LIN {X 0,Y 239.428,Z 683.696,A -85,B 0,C 180,E1 8082.611,E2 8082.611} C_VEL
LIN {X 0,Y 240.054,Z 699.149,A -85,B 0,C 180,E1 8081.155,E2 8081.155} C_VEL
LIN {X 0,Y 233.053,Z 774.476,A -85,B 0,C 180,E1 8079.078,E2 8079.078} C_VEL
LIN {X 0,Y 230.461,Z 791.009,A -85,B 0,C 180,E1 8078.257,E2 8078.257} C_VEL
LIN {X 0,Y 226.592,Z 807.31,A -85,B 0,C 180,E1 8077.072,E2 8077.072} C_VEL
LIN {X 0,Y 221.78,Z 822.279,A -85,B 0,C 180,E1 8075.581,E2 8075.581} C_VEL
LIN {X 0,Y 215.863,Z 836.74,A -85,B 0,C 180,E1 8073.655,E2 8073.655} C_VEL
LIN {X 0,Y 209.493,Z 849.592,A -85,B 0,C 180,E1 8071.408,E2 8071.408} C_VEL
LIN {X 0,Y 202.485,Z 861.469,A -85,B 0,C 180,E1 8068.664,E2 8068.664} C_VEL
LIN {X 0,Y 195.095,Z 872.265,A -85,B 0,C 180,E1 8065.327,E2 8065.327} C_VEL
LIN {X 0,Y 188.35,Z 880.818,A -85,B 0,C 180,E1 8061.77,E2 8061.77} C_VEL
LIN {X 0,Y 181.644,Z 888.195,A -85,B 0,C 180,E1 8057.516,E2 8057.516} C_VEL
LIN {X 0,Y 175.57,Z 894.029,A -85,B 0,C 180,E1 8052.654,E2 8052.654} C_VEL
LIN {X 0,Y 170.723,Z 897.867,A -85,B 0,C 180,E1 8047.515,E2 8047.515} C_VEL
LIN {X 0,Y 166.949,Z 900.056,A -85,B 0,C 180,E1 8041.739,E2 8041.739} C_VEL
LIN {X 0,Y 164.662,Z 900.334,A -85,B 0,C 180,E1 8035.918,E2 8035.918} C_VEL
LIN {X 0,Y 163.665,Z 898.731,A -85,B 0,C 180,E1 8029.809,E2 8029.809} C_VEL
LIN {X 0,Y 163.914,Z 895.477,A -85,B 0,C 180,E1 8024.093,E2 8024.093} C_VEL
LIN {X 0,Y 165.328,Z 890.237,A -85,B 0,C 180,E1 8018.341,E2 8018.341} C_VEL
LIN {X 0,Y 167.764,Z 883.453,A -85,B 0,C 180,E1 8013.07,E2 8013.07} C_VEL
LIN {X 0,Y 171.056,Z 875.039,A -85,B 0,C 180,E1 8008.273,E2 8008.273} C_VEL
LIN {X 0,Y 174.923,Z 865.341,A -85,B 0,C 180,E1 8004.041,E2 8004.041} C_VEL
LIN {X 0,Y 179.081,Z 854.36,A -85,B 0,C 180,E1 8000.354,E2 8000.354} C_VEL
LIN {X 0,Y 183.652,Z 841.158,A -85,B 0,C 180,E1 7996.939,E2 7996.939} C_VEL
LIN {X 0,Y 187.804,Z 827.496,A -85,B 0,C 180,E1 7994.243,E2 7994.243} C_VEL
LIN {X 0,Y 191.755,Z 811.933,A -85,B 0,C 180,E1 7991.924,E2 7991.924} C_VEL
LIN {X 0,Y 194.868,Z 796.193,A -85,B 0,C 180,E1 7990.204,E2 7990.204} C_VEL
LIN {X 0,Y 197.282,Z 778.863,A -85,B 0,C 180,E1 7988.888,E2 7988.888} C_VEL
LIN {X 0,Y 198.697,Z 760.857,A -85,B 0,C 180,E1 7988.063,E2 7988.063} C_VEL
LIN {X 0,Y 203.572,Z 686.601,A -85,B 0,C 180,E1 7985.632,E2 7985.632} C_VEL
LIN {X 0,Y 199.817,Z 646.699,A -85,B 0,C 180,E1 7982.617,E2 7982.617} C_VEL
LIN {X 0,Y 192.297,Z 631.171,A -85,B 0,C 180,E1 7979.45,E2 7979.45} C_VEL
LIN {X 0,Y 189.561,Z 625.909,A -85,B 0,C 180,E1 7978.127,E2 7978.127} C_VEL
LIN {X 0,Y 187.323,Z 616.123,A -85,B 0,C 180,E1 7973.193,E2 7973.193} C_VEL
LIN {X 0,Y 184.89,Z 607.378,A -85,B 0,C 180,E1 7967.888,E2 7967.888} C_VEL
LIN {X 0,Y 182.856,Z 600.739,A -85,B 0,C 180,E1 7963.119,E2 7963.119} C_VEL
LIN {X 0,Y 180.838,Z 594.707,A -85,B 0,C 180,E1 7957.86,E2 7957.86} C_VEL
LIN {X 0,Y 179.177,Z 590.553,A -85,B 0,C 180,E1 7953.153,E2 7953.153} C_VEL
LIN {X 0,Y 177.959,Z 587.255,A -85,B 0,C 180,E1 7948.528,E2 7948.528} C_VEL
LIN {X 0,Y 176.637,Z 583.641,A -85,B 0,C 180,E1 7940.546,E2 7940.546} C_VEL
LIN {X 0,Y 176.092,Z 582.922,A -85,B 0,C 180,E1 7934.133,E2 7934.133} C_VEL
LIN {X 0,Y 176.584,Z 583.469,A -85,B 0,C 180,E1 7927.484,E2 7927.484} C_VEL
LIN {X 0,Y 177.159,Z 584.592,A -85,B 0,C 180,E1 7923.884,E2 7923.884} C_VEL
LIN {X 0,Y 179.034,Z 588.581,A -85,B 0,C 180,E1 7916.479,E2 7916.479} C_VEL
LIN {X 0,Y 180.799,Z 592.823,A -85,B 0,C 180,E1 7911.413,E2 7911.413} C_VEL
LIN {X 0,Y 182.534,Z 597.114,A -85,B 0,C 180,E1 7907.344,E2 7907.344} C_VEL
LIN {X 0,Y 185.067,Z 603.482,A -85,B 0,C 180,E1 7902.39,E2 7902.39} C_VEL
LIN {X 0,Y 188.02,Z 611.83,A -85,B 0,C 180,E1 7897.158,E2 7897.158} C_VEL
LIN {X 0,Y 191.069,Z 621.45,A -85,B 0,C 180,E1 7892.243,E2 7892.243} C_VEL
LIN {X 0,Y 198.28,Z 634.127,A -85,B 0,C 180,E1 7889.131,E2 7889.131} C_VEL
LIN {X 0,Y 205.837,Z 648.788,A -85,B 0,C 180,E1 7886.25,E2 7886.25} C_VEL
LIN {X 0,Y 208.597,Z 655.147,A -85,B 0,C 180,E1 7885.223,E2 7885.223} C_VEL
LIN {X 0,Y 208.82,Z 667.164,A -85,B 0,C 180,E1 7884.604,E2 7884.604} C_VEL
LIN {X 0,Y 203.561,Z 748.117,A -85,B 0,C 180,E1 7882.187,E2 7882.187} C_VEL
LIN {X 0,Y 202.351,Z 755.783,A -85,B 0,C 180,E1 7882.134,E2 7882.134} C_VEL
LIN {X 0,Y 196.3,Z 776.069,A -85,B 0,C 180,E1 7882.677,E2 7882.677} C_VEL
LIN {X 0,Y 195.302,Z 782.654,A -85,B 0,C 180,E1 7882.62,E2 7882.62} C_VEL
LIN {X 0,Y 193.611,Z 802.35,A -85,B 0,C 180,E1 7881.852,E2 7881.852} C_VEL
LIN {X 0,Y 190.848,Z 819.979,A -85,B 0,C 180,E1 7880.72,E2 7880.72} C_VEL
LIN {X 0,Y 186.92,Z 837.364,A -85,B 0,C 180,E1 7879.124,E2 7879.124} C_VEL
LIN {X 0,Y 182.366,Z 853.624,A -85,B 0,C 180,E1 7877.058,E2 7877.058} C_VEL
LIN {X 0,Y 177.233,Z 869.3,A -85,B 0,C 180,E1 7874.391,E2 7874.391} C_VEL
LIN {X 0,Y 171.883,Z 883.863,A -85,B 0,C 180,E1 7871.098,E2 7871.098} C_VEL
LIN {X 0,Y 166.529,Z 897.391,A -85,B 0,C 180,E1 7867.116,E2 7867.116} C_VEL
LIN {X 0,Y 161.793,Z 909.403,A -85,B 0,C 180,E1 7862.526,E2 7862.526} C_VEL
LIN {X 0,Y 158.011,Z 919.598,A -85,B 0,C 180,E1 7857.514,E2 7857.514} C_VEL
LIN {X 0,Y 155.289,Z 928.39,A -85,B 0,C 180,E1 7851.931,E2 7851.931} C_VEL
LIN {X 0,Y 153.926,Z 935.715,A -85,B 0,C 180,E1 7845.835,E2 7845.835} C_VEL
LIN {X 0,Y 154.037,Z 941.459,A -85,B 0,C 180,E1 7839.343,E2 7839.343} C_VEL
LIN {X 0,Y 155.114,Z 944.871,A -85,B 0,C 180,E1 7833.7,E2 7833.7} C_VEL
LIN {X 0,Y 155.742,Z 946.247,A -85,B 0,C 180,E1 7830.004,E2 7830.004} C_VEL
LIN {X 0,Y 154.8,Z 946.748,A -85,B 0,C 180,E1 7825.931,E2 7825.931} C_VEL
LIN {X 0,Y 153.503,Z 945.982,A -85,B 0,C 180,E1 7819.497,E2 7819.497} C_VEL
LIN {X 0,Y 153.729,Z 943.404,A -85,B 0,C 180,E1 7812.598,E2 7812.598} C_VEL
LIN {X 0,Y 155.999,Z 939.047,A -85,B 0,C 180,E1 7805.79,E2 7805.79} C_VEL
LIN {X 0,Y 160.423,Z 932.831,A -85,B 0,C 180,E1 7799.272,E2 7799.272} C_VEL
LIN {X 0,Y 166.479,Z 925.115,A -85,B 0,C 180,E1 7793.526,E2 7793.526} C_VEL
LIN {X 0,Y 173.691,Z 915.929,A -85,B 0,C 180,E1 7788.557,E2 7788.557} C_VEL
LIN {X 0,Y 181.69,Z 905.294,A -85,B 0,C 180,E1 7784.334,E2 7784.334} C_VEL
LIN {X 0,Y 190.524,Z 892.551,A -85,B 0,C 180,E1 7780.597,E2 7780.597} C_VEL
LIN {X 0,Y 198.904,Z 879.059,A -85,B 0,C 180,E1 7777.665,E2 7777.665} C_VEL
LIN {X 0,Y 206.592,Z 864.904,A -85,B 0,C 180,E1 7775.376,E2 7775.376} C_VEL
LIN {X 0,Y 213.561,Z 849.877,A -85,B 0,C 180,E1 7773.567,E2 7773.567} C_VEL
LIN {X 0,Y 219.656,Z 834.019,A -85,B 0,C 180,E1 7772.164,E2 7772.164} C_VEL
LIN {X 0,Y 224.755,Z 817.067,A -85,B 0,C 180,E1 7771.078,E2 7771.078} C_VEL
LIN {X 0,Y 228.519,Z 799.346,A -85,B 0,C 180,E1 7770.277,E2 7770.277} C_VEL
LIN {X 0,Y 230.844,Z 779.683,A -85,B 0,C 180,E1 7769.691,E2 7769.691} C_VEL
LIN {X 0,Y 239.232,Z 685.969,A -85,B 0,C 180,E1 7767.302,E2 7767.302} C_VEL
LIN {X 0,Y 234.919,Z 677.468,A -85,B 0,C 180,E1 7764.116,E2 7764.116} C_VEL
LIN {X 0,Y 231.392,Z 671.367,A -85,B 0,C 180,E1 7761.017,E2 7761.017} C_VEL
LIN {X 0,Y 228.729,Z 667.122,A -85,B 0,C 180,E1 7758.213,E2 7758.213} C_VEL
LIN {X 0,Y 226.198,Z 663.254,A -85,B 0,C 180,E1 7754.724,E2 7754.724} C_VEL
LIN {X 0,Y 224.164,Z 660.314,A -85,B 0,C 180,E1 7750.537,E2 7750.537} C_VEL
LIN {X 0,Y 223.09,Z 659.552,A -85,B 0,C 180,E1 7744.884,E2 7744.884} C_VEL
LIN {X 0,Y 223.271,Z 660.346,A -85,B 0,C 180,E1 7742.309,E2 7742.309} C_VEL
LIN {X 0,Y 224.694,Z 663.258,A -85,B 0,C 180,E1 7737.449,E2 7737.449} C_VEL
LIN {X 0,Y 227.153,Z 668.305,A -85,B 0,C 180,E1 7733.174,E2 7733.174} C_VEL
LIN {X 0,Y 229.056,Z 672.328,A -85,B 0,C 180,E1 7730.705,E2 7730.705} C_VEL
LIN {X 0,Y 231.536,Z 677.558,A -85,B 0,C 180,E1 7728.1,E2 7728.1} C_VEL
LIN {X 0,Y 234.13,Z 683.469,A -85,B 0,C 180,E1 7725.722,E2 7725.722} C_VEL
LIN {X 0,Y 236.21,Z 688.871,A -85,B 0,C 180,E1 7723.982,E2 7723.982} C_VEL
LIN {X 0,Y 236.518,Z 700.902,A -85,B 0,C 180,E1 7722.858,E2 7722.858} C_VEL
LIN {X 0,Y 229.387,Z 775.054,A -85,B 0,C 180,E1 7720.834,E2 7720.834} C_VEL
LIN {X 0,Y 226.705,Z 791.601,A -85,B 0,C 180,E1 7720.023,E2 7720.023} C_VEL
LIN {X 0,Y 222.69,Z 807.951,A -85,B 0,C 180,E1 7718.85,E2 7718.85} C_VEL
LIN {X 0,Y 217.695,Z 822.98,A -85,B 0,C 180,E1 7717.375,E2 7717.375} C_VEL
LIN {X 0,Y 211.543,Z 837.477,A -85,B 0,C 180,E1 7715.465,E2 7715.465} C_VEL
LIN {X 0,Y 204.564,Z 850.981,A -85,B 0,C 180,E1 7713.11,E2 7713.11} C_VEL
LIN {X 0,Y 197.162,Z 862.876,A -85,B 0,C 180,E1 7710.331,E2 7710.331} C_VEL
LIN {X 0,Y 189.505,Z 873.477,A -85,B 0,C 180,E1 7707.011,E2 7707.011} C_VEL
LIN {X 0,Y 182.068,Z 882.342,A -85,B 0,C 180,E1 7703.23,E2 7703.23} C_VEL
LIN {X 0,Y 175.061,Z 889.586,A -85,B 0,C 180,E1 7698.919,E2 7698.919} C_VEL
LIN {X 0,Y 168.617,Z 895.358,A -85,B 0,C 180,E1 7693.92,E2 7693.92} C_VEL
LIN {X 0,Y 163.251,Z 899.255,A -85,B 0,C 180,E1 7688.374,E2 7688.374} C_VEL
LIN {X 0,Y 159.396,Z 901.278,A -85,B 0,C 180,E1 7682.639,E2 7682.639} C_VEL
LIN {X 0,Y 156.986,Z 901.582,A -85,B 0,C 180,E1 7676.878,E2 7676.878} C_VEL
LIN {X 0,Y 155.776,Z 900.032,A -85,B 0,C 180,E1 7670.425,E2 7670.425} C_VEL
LIN {X 0,Y 155.924,Z 896.909,A -85,B 0,C 180,E1 7664.465,E2 7664.465} C_VEL
LIN {X 0,Y 157.191,Z 892.148,A -85,B 0,C 180,E1 7658.776,E2 7658.776} C_VEL
LIN {X 0,Y 159.593,Z 885.6,A -85,B 0,C 180,E1 7653.228,E2 7653.228} C_VEL
LIN {X 0,Y 162.875,Z 877.634,A -85,B 0,C 180,E1 7648.237,E2 7648.237} C_VEL
LIN {X 0,Y 167.129,Z 867.453,A -85,B 0,C 180,E1 7643.47,E2 7643.47} C_VEL
LIN {X 0,Y 171.691,Z 856.124,A -85,B 0,C 180,E1 7639.426,E2 7639.426} C_VEL
LIN {X 0,Y 176.451,Z 843.081,A -85,B 0,C 180,E1 7635.895,E2 7635.895} C_VEL
LIN {X 0,Y 180.761,Z 829.784,A -85,B 0,C 180,E1 7633.126,E2 7633.126} C_VEL
LIN {X 0,Y 184.887,Z 814.509,A -85,B 0,C 180,E1 7630.736,E2 7630.736} C_VEL
LIN {X 0,Y 188.268,Z 798.796,A -85,B 0,C 180,E1 7628.91,E2 7628.91} C_VEL
LIN {X 0,Y 190.822,Z 781.973,A -85,B 0,C 180,E1 7627.55,E2 7627.55} C_VEL
LIN {X 0,Y 192.42,Z 764.7,A -85,B 0,C 180,E1 7626.667,E2 7626.667} C_VEL
LIN {X 0,Y 197.669,Z 687.648,A -85,B 0,C 180,E1 7624.1,E2 7624.1} C_VEL
LIN {X 0,Y 194.418,Z 650.352,A -85,B 0,C 180,E1 7621.19,E2 7621.19} C_VEL
LIN {X 0,Y 187.727,Z 636.24,A -85,B 0,C 180,E1 7618.161,E2 7618.161} C_VEL
LIN {X 0,Y 182.096,Z 625.601,A -85,B 0,C 180,E1 7615.284,E2 7615.284} C_VEL
LIN {X 0,Y 180.173,Z 617.536,A -85,B 0,C 180,E1 7610.754,E2 7610.754} C_VEL
LIN {X 0,Y 178.21,Z 610.241,A -85,B 0,C 180,E1 7605.903,E2 7605.903} C_VEL
LIN {X 0,Y 176.352,Z 604.108,A -85,B 0,C 180,E1 7601.056,E2 7601.056} C_VEL
LIN {X 0,Y 174.761,Z 599.428,A -85,B 0,C 180,E1 7596.514,E2 7596.514} C_VEL
LIN {X 0,Y 173.64,Z 596.234,A -85,B 0,C 180,E1 7592.771,E2 7592.771} C_VEL
LIN {X 0,Y 172.573,Z 593.132,A -85,B 0,C 180,E1 7588.278,E2 7588.278} C_VEL
LIN {X 0,Y 171.434,Z 589.715,A -85,B 0,C 180,E1 7580.484,E2 7580.484} C_VEL
LIN {X 0,Y 170.944,Z 589.036,A -85,B 0,C 180,E1 7573.85,E2 7573.85} C_VEL
LIN {X 0,Y 171.464,Z 589.628,A -85,B 0,C 180,E1 7567.371,E2 7567.371} C_VEL
LIN {X 0,Y 171.97,Z 590.687,A -85,B 0,C 180,E1 7564.001,E2 7564.001} C_VEL
LIN {X 0,Y 173.71,Z 594.549,A -85,B 0,C 180,E1 7556.701,E2 7556.701} C_VEL
LIN {X 0,Y 175.407,Z 598.878,A -85,B 0,C 180,E1 7551.478,E2 7551.478} C_VEL
LIN {X 0,Y 176.998,Z 602.87,A -85,B 0,C 180,E1 7547.605,E2 7547.605} C_VEL
LIN {X 0,Y 179.299,Z 608.874,A -85,B 0,C 180,E1 7542.81,E2 7542.81} C_VEL
LIN {X 0,Y 182.117,Z 617.308,A -85,B 0,C 180,E1 7537.399,E2 7537.399} C_VEL
LIN {X 0,Y 183.778,Z 622.203,A -85,B 0,C 180,E1 7534.847,E2 7534.847} C_VEL
LIN {X 0,Y 190.897,Z 634.308,A -85,B 0,C 180,E1 7531.492,E2 7531.492} C_VEL
LIN {X 0,Y 198.02,Z 647.764,A -85,B 0,C 180,E1 7528.494,E2 7528.494} C_VEL
LIN {X 0,Y 202.815,Z 658.233,A -85,B 0,C 180,E1 7526.602,E2 7526.602} C_VEL
LIN {X 0,Y 202.909,Z 668.079,A -85,B 0,C 180,E1 7526.097,E2 7526.097} C_VEL
LIN {X 0,Y 195.302,Z 782.654,A -85,B 0,C 180,E1 7522.62,E2 7522.62} C_VEL
LIN {X 0,Y 193.966,Z 790.299,A -85,B 0,C 180,E1 7522.569,E2 7522.569} C_VEL
LIN {X 0,Y 187.888,Z 807.129,A -85,B 0,C 180,E1 7522.822,E2 7522.822} C_VEL
LIN {X 0,Y 185.613,Z 814.554,A -85,B 0,C 180,E1 7522.604,E2 7522.604} C_VEL
LIN {X 0,Y 185.173,Z 816.696,A -85,B 0,C 180,E1 7522.471,E2 7522.471} C_VEL
LIN {X 0,Y 181.426,Z 833.575,A -85,B 0,C 180,E1 7520.993,E2 7520.993} C_VEL
LIN {X 0,Y 176.881,Z 849.68,A -85,B 0,C 180,E1 7519.027,E2 7519.027} C_VEL
LIN {X 0,Y 171.432,Z 866.024,A -85,B 0,C 180,E1 7516.321,E2 7516.321} C_VEL
LIN {X 0,Y 165.984,Z 880.498,A -85,B 0,C 180,E1 7513.135,E2 7513.135} C_VEL
LIN {X 0,Y 160.473,Z 893.91,A -85,B 0,C 180,E1 7509.263,E2 7509.263} C_VEL
LIN {X 0,Y 155.217,Z 906.376,A -85,B 0,C 180,E1 7504.534,E2 7504.534} C_VEL
LIN {X 0,Y 150.738,Z 917.592,A -85,B 0,C 180,E1 7498.964,E2 7498.964} C_VEL
LIN {X 0,Y 147.585,Z 926.935,A -85,B 0,C 180,E1 7492.874,E2 7492.874} C_VEL
LIN {X 0,Y 146.01,Z 934.479,A -85,B 0,C 180,E1 7486.309,E2 7486.309} C_VEL
LIN {X 0,Y 146.075,Z 940.247,A -85,B 0,C 180,E1 7479.459,E2 7479.459} C_VEL
LIN {X 0,Y 147.236,Z 943.726,A -85,B 0,C 180,E1 7473.396,E2 7473.396} C_VEL
LIN {X 0,Y 147.844,Z 944.945,A -85,B 0,C 180,E1 7470.005,E2 7470.005} C_VEL
LIN {X 0,Y 146.798,Z 945.483,A -85,B 0,C 180,E1 7465.708,E2 7465.708} C_VEL
LIN {X 0,Y 145.507,Z 944.797,A -85,B 0,C 180,E1 7458.913,E2 7458.913} C_VEL
LIN {X 0,Y 145.924,Z 942.317,A -85,B 0,C 180,E1 7451.635,E2 7451.635} C_VEL
LIN {X 0,Y 148.597,Z 937.956,A -85,B 0,C 180,E1 7444.373,E2 7444.373} C_VEL
LIN {X 0,Y 153.745,Z 931.538,A -85,B 0,C 180,E1 7437.34,E2 7437.34} C_VEL
LIN {X 0,Y 160.388,Z 923.803,A -85,B 0,C 180,E1 7431.445,E2 7431.445} C_VEL
LIN {X 0,Y 168.168,Z 914.58,A -85,B 0,C 180,E1 7426.405,E2 7426.405} C_VEL
LIN {X 0,Y 176.691,Z 903.905,A -85,B 0,C 180,E1 7422.169,E2 7422.169} C_VEL
LIN {X 0,Y 185.532,Z 891.794,A -85,B 0,C 180,E1 7418.621,E2 7418.621} C_VEL
LIN {X 0,Y 194.07,Z 878.728,A -85,B 0,C 180,E1 7415.775,E2 7415.775} C_VEL
LIN {X 0,Y 202.41,Z 864.08,A -85,B 0,C 180,E1 7413.417,E2 7413.417} C_VEL
LIN {X 0,Y 209.646,Z 849.014,A -85,B 0,C 180,E1 7411.642,E2 7411.642} C_VEL
LIN {X 0,Y 216.304,Z 832.104,A -85,B 0,C 180,E1 7410.2,E2 7410.2} C_VEL
LIN {X 0,Y 221.507,Z 814.966,A -85,B 0,C 180,E1 7409.155,E2 7409.155} C_VEL
LIN {X 0,Y 225.181,Z 797.447,A -85,B 0,C 180,E1 7408.407,E2 7408.407} C_VEL
LIN {X 0,Y 227.613,Z 776.617,A -85,B 0,C 180,E1 7407.814,E2 7407.814} C_VEL
LIN {X 0,Y 235.634,Z 690.369,A -85,B 0,C 180,E1 7405.646,E2 7405.646} C_VEL
LIN {X 0,Y 232.101,Z 683.326,A -85,B 0,C 180,E1 7402.745,E2 7402.745} C_VEL
LIN {X 0,Y 229.499,Z 678.565,A -85,B 0,C 180,E1 7400.264,E2 7400.264} C_VEL
LIN {X 0,Y 227.206,Z 674.687,A -85,B 0,C 180,E1 7397.676,E2 7397.676} C_VEL
LIN {X 0,Y 224.807,Z 670.838,A -85,B 0,C 180,E1 7394.159,E2 7394.159} C_VEL
LIN {X 0,Y 223.066,Z 668.204,A -85,B 0,C 180,E1 7390.328,E2 7390.328} C_VEL
LIN {X 0,Y 222.072,Z 667.487,A -85,B 0,C 180,E1 7384.907,E2 7384.907} C_VEL
LIN {X 0,Y 222.245,Z 668.339,A -85,B 0,C 180,E1 7382.32,E2 7382.32} C_VEL
LIN {X 0,Y 223.477,Z 671.041,A -85,B 0,C 180,E1 7377.82,E2 7377.82} C_VEL
LIN {X 0,Y 225.984,Z 676.519,A -85,B 0,C 180,E1 7373.266,E2 7373.266} C_VEL
LIN {X 0,Y 229.211,Z 683.798,A -85,B 0,C 180,E1 7369.252,E2 7369.252} C_VEL
LIN {X 0,Y 231.879,Z 690.276,A -85,B 0,C 180,E1 7366.598,E2 7366.598} C_VEL
LIN {X 0,Y 233.168,Z 694.083,A -85,B 0,C 180,E1 7365.392,E2 7365.392} C_VEL
LIN {X 0,Y 233.222,Z 702.547,A -85,B 0,C 180,E1 7364.616,E2 7364.616} C_VEL
LIN {X 0,Y 225.919,Z 775.846,A -85,B 0,C 180,E1 7362.638,E2 7362.638} C_VEL
LIN {X 0,Y 223.123,Z 792.417,A -85,B 0,C 180,E1 7361.834,E2 7361.834} C_VEL
LIN {X 0,Y 219.01,Z 808.593,A -85,B 0,C 180,E1 7360.691,E2 7360.691} C_VEL
LIN {X 0,Y 213.833,Z 823.681,A -85,B 0,C 180,E1 7359.235,E2 7359.235} C_VEL
LIN {X 0,Y 207.815,Z 837.452,A -85,B 0,C 180,E1 7357.462,E2 7357.462} C_VEL
LIN {X 0,Y 200.533,Z 851.132,A -85,B 0,C 180,E1 7355.136,E2 7355.136} C_VEL
LIN {X 0,Y 192.876,Z 863.101,A -85,B 0,C 180,E1 7352.414,E2 7352.414} C_VEL
LIN {X 0,Y 184.641,Z 874.043,A -85,B 0,C 180,E1 7349.039,E2 7349.039} C_VEL
LIN {X 0,Y 176.614,Z 883.204,A -85,B 0,C 180,E1 7345.159,E2 7345.159} C_VEL
LIN {X 0,Y 169.074,Z 890.559,A -85,B 0,C 180,E1 7340.744,E2 7340.744} C_VEL
LIN {X 0,Y 162.169,Z 896.359,A -85,B 0,C 180,E1 7335.648,E2 7335.648} C_VEL
LIN {X 0,Y 156.541,Z 900.223,A -85,B 0,C 180,E1 7330.163,E2 7330.163} C_VEL
LIN {X 0,Y 152.077,Z 902.425,A -85,B 0,C 180,E1 7323.967,E2 7323.967} C_VEL
LIN {X 0,Y 149.222,Z 902.777,A -85,B 0,C 180,E1 7317.53,E2 7317.53} C_VEL
LIN {X 0,Y 147.892,Z 901.292,A -85,B 0,C 180,E1 7310.99,E2 7310.99} C_VEL
LIN {X 0,Y 147.981,Z 898.065,A -85,B 0,C 180,E1 7304.471,E2 7304.471} C_VEL
LIN {X 0,Y 149.299,Z 893.282,A -85,B 0,C 180,E1 7298.467,E2 7298.467} C_VEL
LIN {X 0,Y 151.823,Z 886.728,A -85,B 0,C 180,E1 7292.637,E2 7292.637} C_VEL
LIN {X 0,Y 155.28,Z 878.768,A -85,B 0,C 180,E1 7287.412,E2 7287.412} C_VEL
LIN {X 0,Y 159.755,Z 868.601,A -85,B 0,C 180,E1 7282.444,E2 7282.444} C_VEL
LIN {X 0,Y 164.546,Z 857.31,A -85,B 0,C 180,E1 7278.251,E2 7278.251} C_VEL
LIN {X 0,Y 169.536,Z 844.313,A -85,B 0,C 180,E1 7274.607,E2 7274.607} C_VEL
LIN {X 0,Y 174.306,Z 830.259,A -85,B 0,C 180,E1 7271.607,E2 7271.607} C_VEL
LIN {X 0,Y 178.532,Z 815.274,A -85,B 0,C 180,E1 7269.221,E2 7269.221} C_VEL
LIN {X 0,Y 182.019,Z 799.792,A -85,B 0,C 180,E1 7267.384,E2 7267.384} C_VEL
LIN {X 0,Y 184.711,Z 783,A -85,B 0,C 180,E1 7265.992,E2 7265.992} C_VEL
LIN {X 0,Y 186.42,Z 765.577,A -85,B 0,C 180,E1 7265.077,E2 7265.077} C_VEL
LIN {X 0,Y 191.894,Z 688.725,A -85,B 0,C 180,E1 7262.487,E2 7262.487} C_VEL
LIN {X 0,Y 189.113,Z 653.977,A -85,B 0,C 180,E1 7259.67,E2 7259.67} C_VEL
LIN {X 0,Y 183.183,Z 641.172,A -85,B 0,C 180,E1 7256.772,E2 7256.772} C_VEL
LIN {X 0,Y 177.12,Z 629.878,A -85,B 0,C 180,E1 7253.556,E2 7253.556} C_VEL
LIN {X 0,Y 174.72,Z 625.277,A -85,B 0,C 180,E1 7252.014,E2 7252.014} C_VEL
LIN {X 0,Y 172.617,Z 616.63,A -85,B 0,C 180,E1 7246.39,E2 7246.39} C_VEL
LIN {X 0,Y 170.67,Z 609.919,A -85,B 0,C 180,E1 7241.008,E2 7241.008} C_VEL
LIN {X 0,Y 169.18,Z 605.096,A -85,B 0,C 180,E1 7236.229,E2 7236.229} C_VEL
LIN {X 0,Y 168.116,Z 601.918,A -85,B 0,C 180,E1 7232.363,E2 7232.363} C_VEL
LIN {X 0,Y 167.151,Z 598.936,A -85,B 0,C 180,E1 7227.813,E2 7227.813} C_VEL
LIN {X 0,Y 166.189,Z 595.721,A -85,B 0,C 180,E1 7220.057,E2 7220.057} C_VEL
LIN {X 0,Y 165.791,Z 595.169,A -85,B 0,C 180,E1 7213.249,E2 7213.249} C_VEL
LIN {X 0,Y 166.394,Z 595.862,A -85,B 0,C 180,E1 7206.903,E2 7206.903} C_VEL
LIN {X 0,Y 166.809,Z 596.944,A -85,B 0,C 180,E1 7203.781,E2 7203.781} C_VEL
LIN {X 0,Y 168.383,Z 600.51,A -85,B 0,C 180,E1 7196.937,E2 7196.937} C_VEL
LIN {X 0,Y 169.935,Z 604.59,A -85,B 0,C 180,E1 7191.883,E2 7191.883} C_VEL
LIN {X 0,Y 171.578,Z 608.986,A -85,B 0,C 180,E1 7187.549,E2 7187.549} C_VEL
LIN {X 0,Y 173.801,Z 615.184,A -85,B 0,C 180,E1 7182.594,E2 7182.594} C_VEL
LIN {X 0,Y 176.223,Z 622.331,A -85,B 0,C 180,E1 7178.042,E2 7178.042} C_VEL
LIN {X 0,Y 183.415,Z 634.045,A -85,B 0,C 180,E1 7174.232,E2 7174.232} C_VEL
LIN {X 0,Y 190.901,Z 647.915,A -85,B 0,C 180,E1 7170.722,E2 7170.722} C_VEL
LIN {X 0,Y 197.123,Z 661.227,A -85,B 0,C 180,E1 7168.057,E2 7168.057} C_VEL
LIN {X 0,Y 197.091,Z 669.084,A -85,B 0,C 180,E1 7167.663,E2 7167.663} C_VEL
LIN {X 0,Y 188.187,Z 795.645,A -85,B 0,C 180,E1 7163.7,E2 7163.7} C_VEL
LIN {X 0,Y 185.672,Z 813.843,A -85,B 0,C 180,E1 7162.668,E2 7162.668} C_VEL
LIN {X 0,Y 185.173,Z 816.696,A -85,B 0,C 180,E1 7162.471,E2 7162.471} C_VEL
LIN {X 0,Y 182.945,Z 824.046,A -85,B 0,C 180,E1 7162.105,E2 7162.105} C_VEL
LIN {X 0,Y 175.698,Z 837.88,A -85,B 0,C 180,E1 7161.662,E2 7161.662} C_VEL
LIN {X 0,Y 171.758,Z 845.678,A -85,B 0,C 180,E1 7161.063,E2 7161.063} C_VEL
LIN {X 0,Y 170.648,Z 848.607,A -85,B 0,C 180,E1 7160.685,E2 7160.685} C_VEL
LIN {X 0,Y 164.976,Z 864.953,A -85,B 0,C 180,E1 7157.939,E2 7157.939} C_VEL
LIN {X 0,Y 159.271,Z 879.456,A -85,B 0,C 180,E1 7154.678,E2 7154.678} C_VEL
LIN {X 0,Y 153.446,Z 892.977,A -85,B 0,C 180,E1 7150.664,E2 7150.664} C_VEL
LIN {X 0,Y 147.933,Z 905.347,A -85,B 0,C 180,E1 7145.801,E2 7145.801} C_VEL
LIN {X 0,Y 143.197,Z 916.499,A -85,B 0,C 180,E1 7140.025,E2 7140.025} C_VEL
LIN {X 0,Y 139.803,Z 925.856,A -85,B 0,C 180,E1 7133.613,E2 7133.613} C_VEL
LIN {X 0,Y 138.105,Z 933.243,A -85,B 0,C 180,E1 7126.837,E2 7126.837} C_VEL
LIN {X 0,Y 138.067,Z 938.775,A -85,B 0,C 180,E1 7119.977,E2 7119.977} C_VEL
LIN {X 0,Y 139.305,Z 942.479,A -85,B 0,C 180,E1 7113.296,E2 7113.296} C_VEL
LIN {X 0,Y 139.943,Z 943.641,A -85,B 0,C 180,E1 7110.005,E2 7110.005} C_VEL
LIN {X 0,Y 138.79,Z 944.205,A -85,B 0,C 180,E1 7105.46,E2 7105.46} C_VEL
LIN {X 0,Y 137.522,Z 943.591,A -85,B 0,C 180,E1 7098.26,E2 7098.26} C_VEL
LIN {X 0,Y 138.162,Z 941.225,A -85,B 0,C 180,E1 7090.562,E2 7090.562} C_VEL
LIN {X 0,Y 141.154,Z 937.056,A -85,B 0,C 180,E1 7083.05,E2 7083.05} C_VEL
LIN {X 0,Y 146.524,Z 931.027,A -85,B 0,C 180,E1 7075.984,E2 7075.984} C_VEL
LIN {X 0,Y 153.582,Z 923.48,A -85,B 0,C 180,E1 7069.881,E2 7069.881} C_VEL
LIN {X 0,Y 161.781,Z 914.503,A -85,B 0,C 180,E1 7064.716,E2 7064.716} C_VEL
LIN {X 0,Y 170.699,Z 904.147,A -85,B 0,C 180,E1 7060.419,E2 7060.419} C_VEL
LIN {X 0,Y 179.894,Z 892.32,A -85,B 0,C 180,E1 7056.849,E2 7056.849} C_VEL
LIN {X 0,Y 189.094,Z 878.99,A -85,B 0,C 180,E1 7053.899,E2 7053.899} C_VEL
LIN {X 0,Y 197.709,Z 864.627,A -85,B 0,C 180,E1 7051.569,E2 7051.569} C_VEL
LIN {X 0,Y 205.475,Z 849.294,A -85,B 0,C 180,E1 7049.758,E2 7049.758} C_VEL
LIN {X 0,Y 211.987,Z 833.571,A -85,B 0,C 180,E1 7048.416,E2 7048.416} C_VEL
LIN {X 0,Y 217.692,Z 815.806,A -85,B 0,C 180,E1 7047.329,E2 7047.329} C_VEL
LIN {X 0,Y 221.694,Z 798.062,A -85,B 0,C 180,E1 7046.567,E2 7046.567} C_VEL
LIN {X 0,Y 224.17,Z 778.537,A -85,B 0,C 180,E1 7046.006,E2 7046.006} C_VEL
LIN {X 0,Y 232.275,Z 694.952,A -85,B 0,C 180,E1 7043.942,E2 7043.942} C_VEL
LIN {X 0,Y 229.365,Z 688.987,A -85,B 0,C 180,E1 7041.278,E2 7041.278} C_VEL
LIN {X 0,Y 226.096,Z 682.796,A -85,B 0,C 180,E1 7037.633,E2 7037.633} C_VEL
LIN {X 0,Y 223.435,Z 678.425,A -85,B 0,C 180,E1 7033.587,E2 7033.587} C_VEL
LIN {X 0,Y 221.884,Z 676.025,A -85,B 0,C 180,E1 7029.859,E2 7029.859} C_VEL
LIN {X 0,Y 221.056,Z 675.444,A -85,B 0,C 180,E1 7024.669,E2 7024.669} C_VEL
LIN {X 0,Y 221.768,Z 677.715,A -85,B 0,C 180,E1 7019.741,E2 7019.741} C_VEL
LIN {X 0,Y 222.693,Z 679.871,A -85,B 0,C 180,E1 7017.169,E2 7017.169} C_VEL
LIN {X 0,Y 225.1,Z 685.504,A -85,B 0,C 180,E1 7012.919,E2 7012.919} C_VEL
LIN {X 0,Y 227.509,Z 691.459,A -85,B 0,C 180,E1 7009.804,E2 7009.804} C_VEL
LIN {X 0,Y 229.992,Z 697.879,A -85,B 0,C 180,E1 7007.19,E2 7007.19} C_VEL
LIN {X 0,Y 230.274,Z 699.095,A -85,B 0,C 180,E1 7006.871,E2 7006.871} C_VEL
LIN {X 0,Y 230.212,Z 704.154,A -85,B 0,C 180,E1 7006.429,E2 7006.429} C_VEL
LIN {X 0,Y 222.764,Z 776.43,A -85,B 0,C 180,E1 7004.51,E2 7004.51} C_VEL
LIN {X 0,Y 219.853,Z 793.084,A -85,B 0,C 180,E1 7003.716,E2 7003.716} C_VEL
LIN {X 0,Y 215.568,Z 809.329,A -85,B 0,C 180,E1 7002.588,E2 7002.588} C_VEL
LIN {X 0,Y 210.022,Z 824.843,A -85,B 0,C 180,E1 7001.111,E2 7001.111} C_VEL
LIN {X 0,Y 203.195,Z 839.706,A -85,B 0,C 180,E1 6999.194,E2 6999.194} C_VEL
LIN {X 0,Y 195.655,Z 853.141,A -85,B 0,C 180,E1 6996.884,E2 6996.884} C_VEL
LIN {X 0,Y 187.699,Z 864.878,A -85,B 0,C 180,E1 6994.172,E2 6994.172} C_VEL
LIN {X 0,Y 179.52,Z 875.207,A -85,B 0,C 180,E1 6990.96,E2 6990.96} C_VEL
LIN {X 0,Y 171.133,Z 884.3,A -85,B 0,C 180,E1 6987.087,E2 6987.087} C_VEL
LIN {X 0,Y 163.219,Z 891.599,A -85,B 0,C 180,E1 6982.665,E2 6982.665} C_VEL
LIN {X 0,Y 155.888,Z 897.381,A -85,B 0,C 180,E1 6977.516,E2 6977.516} C_VEL
LIN {X 0,Y 149.777,Z 901.319,A -85,B 0,C 180,E1 6971.869,E2 6971.869} C_VEL
LIN {X 0,Y 144.851,Z 903.574,A -85,B 0,C 180,E1 6965.429,E2 6965.429} C_VEL
LIN {X 0,Y 141.626,Z 904.02,A -85,B 0,C 180,E1 6958.682,E2 6958.682} C_VEL
LIN {X 0,Y 140.041,Z 902.607,A -85,B 0,C 180,E1 6951.786,E2 6951.786} C_VEL
LIN {X 0,Y 139.992,Z 899.456,A -85,B 0,C 180,E1 6944.893,E2 6944.893} C_VEL
LIN {X 0,Y 141.281,Z 894.801,A -85,B 0,C 180,E1 6938.541,E2 6938.541} C_VEL
LIN {X 0,Y 143.853,Z 888.346,A -85,B 0,C 180,E1 6932.385,E2 6932.385} C_VEL
LIN {X 0,Y 147.422,Z 880.531,A -85,B 0,C 180,E1 6926.885,E2 6926.885} C_VEL
LIN {X 0,Y 151.702,Z 871.359,A -85,B 0,C 180,E1 6922.04,E2 6922.04} C_VEL
LIN {X 0,Y 156.83,Z 859.946,A -85,B 0,C 180,E1 6917.477,E2 6917.477} C_VEL
LIN {X 0,Y 161.771,Z 848.043,A -85,B 0,C 180,E1 6913.848,E2 6913.848} C_VEL
LIN {X 0,Y 166.929,Z 833.845,A -85,B 0,C 180,E1 6910.581,E2 6910.581} C_VEL
LIN {X 0,Y 171.412,Z 819.425,A -85,B 0,C 180,E1 6908.077,E2 6908.077} C_VEL
LIN {X 0,Y 175.218,Z 804,A -85,B 0,C 180,E1 6906.097,E2 6906.097} C_VEL
LIN {X 0,Y 178.349,Z 786.97,A -85,B 0,C 180,E1 6904.535,E2 6904.535} C_VEL
LIN {X 0,Y 180.304,Z 769.786,A -85,B 0,C 180,E1 6903.529,E2 6903.529} C_VEL
LIN {X 0,Y 186.263,Z 689.601,A -85,B 0,C 180,E1 6900.757,E2 6900.757} C_VEL
LIN {X 0,Y 183.88,Z 657.353,A -85,B 0,C 180,E1 6898.024,E2 6898.024} C_VEL
LIN {X 0,Y 177.415,Z 643.324,A -85,B 0,C 180,E1 6894.595,E2 6894.595} C_VEL
LIN {X 0,Y 171.156,Z 631.574,A -85,B 0,C 180,E1 6890.881,E2 6890.881} C_VEL
LIN {X 0,Y 167.45,Z 625.186,A -85,B 0,C 180,E1 6888.279,E2 6888.279} C_VEL
LIN {X 0,Y 165.791,Z 618.593,A -85,B 0,C 180,E1 6883.435,E2 6883.435} C_VEL
LIN {X 0,Y 164.23,Z 612.926,A -85,B 0,C 180,E1 6878.244,E2 6878.244} C_VEL
LIN {X 0,Y 162.978,Z 608.344,A -85,B 0,C 180,E1 6873.095,E2 6873.095} C_VEL
LIN {X 0,Y 161.816,Z 604.87,A -85,B 0,C 180,E1 6867.609,E2 6867.609} C_VEL
LIN {X 0,Y 160.985,Z 601.793,A -85,B 0,C 180,E1 6859.975,E2 6859.975} C_VEL
LIN {X 0,Y 160.644,Z 601.292,A -85,B 0,C 180,E1 6853.315,E2 6853.315} C_VEL
LIN {X 0,Y 161.267,Z 602.016,A -85,B 0,C 180,E1 6846.766,E2 6846.766} C_VEL
LIN {X 0,Y 161.735,Z 603.545,A -85,B 0,C 180,E1 6842.836,E2 6842.836} C_VEL
LIN {X 0,Y 163.059,Z 606.467,A -85,B 0,C 180,E1 6837.189,E2 6837.189} C_VEL
LIN {X 0,Y 164.479,Z 610.358,A -85,B 0,C 180,E1 6832.246,E2 6832.246} C_VEL
LIN {X 0,Y 166.025,Z 614.707,A -85,B 0,C 180,E1 6827.832,E2 6827.832} C_VEL
LIN {X 0,Y 168.169,Z 621.007,A -85,B 0,C 180,E1 6822.706,E2 6822.706} C_VEL
LIN {X 0,Y 169.157,Z 623.238,A -85,B 0,C 180,E1 6821.476,E2 6821.476} C_VEL
LIN {X 0,Y 174.241,Z 631.179,A -85,B 0,C 180,E1 6818.308,E2 6818.308} C_VEL
LIN {X 0,Y 179.905,Z 640.744,A -85,B 0,C 180,E1 6815.191,E2 6815.191} C_VEL
LIN {X 0,Y 186.612,Z 653.557,A -85,B 0,C 180,E1 6811.869,E2 6811.869} C_VEL
LIN {X 0,Y 191.578,Z 664.589,A -85,B 0,C 180,E1 6809.575,E2 6809.575} C_VEL
LIN {X 0,Y 191.281,Z 672.04,A -85,B 0,C 180,E1 6809.264,E2 6809.264} C_VEL
LIN {X 0,Y 182.246,Z 795.033,A -85,B 0,C 180,E1 6805.363,E2 6805.363} C_VEL
LIN {X 0,Y 179.638,Z 813.21,A -85,B 0,C 180,E1 6804.319,E2 6804.319} C_VEL
LIN {X 0,Y 175.884,Z 830.43,A -85,B 0,C 180,E1 6802.872,E2 6802.872} C_VEL
LIN {X 0,Y 171.241,Z 846.796,A -85,B 0,C 180,E1 6800.948,E2 6800.948} C_VEL
LIN {X 0,Y 170.648,Z 848.607,A -85,B 0,C 180,E1 6800.685,E2 6800.685} C_VEL
LIN {X 0,Y 167.582,Z 855.401,A -85,B 0,C 180,E1 6799.84,E2 6799.84} C_VEL
LIN {X 0,Y 158.341,Z 868.714,A -85,B 0,C 180,E1 6798.325,E2 6798.325} C_VEL
LIN {X 0,Y 153.963,Z 875.608,A -85,B 0,C 180,E1 6797.056,E2 6797.056} C_VEL
LIN {X 0,Y 153.152,Z 877.3,A -85,B 0,C 180,E1 6796.64,E2 6796.64} C_VEL
LIN {X 0,Y 147.064,Z 890.861,A -85,B 0,C 180,E1 6792.603,E2 6792.603} C_VEL
LIN {X 0,Y 141.487,Z 902.704,A -85,B 0,C 180,E1 6787.941,E2 6787.941} C_VEL
LIN {X 0,Y 136.515,Z 913.517,A -85,B 0,C 180,E1 6782.324,E2 6782.324} C_VEL
LIN {X 0,Y 132.487,Z 923.439,A -85,B 0,C 180,E1 6775.482,E2 6775.482} C_VEL
LIN {X 0,Y 130.346,Z 931.186,A -85,B 0,C 180,E1 6768.335,E2 6768.335} C_VEL
LIN {X 0,Y 130.02,Z 936.966,A -85,B 0,C 180,E1 6761.089,E2 6761.089} C_VEL
LIN {X 0,Y 131.193,Z 940.931,A -85,B 0,C 180,E1 6753.938,E2 6753.938} C_VEL
LIN {X 0,Y 132.039,Z 942.337,A -85,B 0,C 180,E1 6750.005,E2 6750.005} C_VEL
LIN {X 0,Y 130.591,Z 942.96,A -85,B 0,C 180,E1 6744.456,E2 6744.456} C_VEL
LIN {X 0,Y 129.532,Z 942.232,A -85,B 0,C 180,E1 6736.552,E2 6736.552} C_VEL
LIN {X 0,Y 130.845,Z 939.55,A -85,B 0,C 180,E1 6728.018,E2 6728.018} C_VEL
LIN {X 0,Y 134.692,Z 935.179,A -85,B 0,C 180,E1 6720.183,E2 6720.183} C_VEL
LIN {X 0,Y 140.99,Z 928.946,A -85,B 0,C 180,E1 6712.94,E2 6712.94} C_VEL
LIN {X 0,Y 148.925,Z 921.199,A -85,B 0,C 180,E1 6706.79,E2 6706.79} C_VEL
LIN {X 0,Y 157.998,Z 911.868,A -85,B 0,C 180,E1 6701.641,E2 6701.641} C_VEL
LIN {X 0,Y 167.534,Z 901.239,A -85,B 0,C 180,E1 6697.475,E2 6697.475} C_VEL
LIN {X 0,Y 177.3,Z 889.063,A -85,B 0,C 180,E1 6694.02,E2 6694.02} C_VEL
LIN {X 0,Y 186.458,Z 876.101,A -85,B 0,C 180,E1 6691.342,E2 6691.342} C_VEL
LIN {X 0,Y 195.205,Z 861.695,A -85,B 0,C 180,E1 6689.17,E2 6689.17} C_VEL
LIN {X 0,Y 202.902,Z 846.57,A -85,B 0,C 180,E1 6687.518,E2 6687.518} C_VEL
LIN {X 0,Y 209.561,Z 830.583,A -85,B 0,C 180,E1 6686.253,E2 6686.253} C_VEL
LIN {X 0,Y 215.037,Z 813.538,A -85,B 0,C 180,E1 6685.28,E2 6685.28} C_VEL
LIN {X 0,Y 218.934,Z 796.01,A -85,B 0,C 180,E1 6684.578,E2 6684.578} C_VEL
LIN {X 0,Y 221.569,Z 774.876,A -85,B 0,C 180,E1 6684.002,E2 6684.002} C_VEL
LIN {X 0,Y 229.075,Z 699.504,A -85,B 0,C 180,E1 6682.133,E2 6682.133} C_VEL
LIN {X 0,Y 226.166,Z 693.508,A -85,B 0,C 180,E1 6679.095,E2 6679.095} C_VEL
LIN {X 0,Y 224.039,Z 689.532,A -85,B 0,C 180,E1 6676.329,E2 6676.329} C_VEL
LIN {X 0,Y 222.084,Z 686.024,A -85,B 0,C 180,E1 6673.009,E2 6673.009} C_VEL
LIN {X 0,Y 220.791,Z 683.916,A -85,B 0,C 180,E1 6669.645,E2 6669.645} C_VEL
LIN {X 0,Y 220.042,Z 683.403,A -85,B 0,C 180,E1 6664.43,E2 6664.43} C_VEL
LIN {X 0,Y 221.051,Z 686.484,A -85,B 0,C 180,E1 6658.704,E2 6658.704} C_VEL
LIN {X 0,Y 223.28,Z 692.126,A -85,B 0,C 180,E1 6654.023,E2 6654.023} C_VEL
LIN {X 0,Y 225.617,Z 698.53,A -85,B 0,C 180,E1 6650.626,E2 6650.626} C_VEL
LIN {X 0,Y 227.53,Z 703.875,A -85,B 0,C 180,E1 6648.418,E2 6648.418} C_VEL
LIN {X 0,Y 227.225,Z 707.8,A -85,B 0,C 180,E1 6648.239,E2 6648.239} C_VEL
LIN {X 0,Y 219.831,Z 777.335,A -85,B 0,C 180,E1 6646.424,E2 6646.424} C_VEL
LIN {X 0,Y 216.778,Z 794.069,A -85,B 0,C 180,E1 6645.637,E2 6645.637} C_VEL
LIN {X 0,Y 212.354,Z 810.248,A -85,B 0,C 180,E1 6644.535,E2 6644.535} C_VEL
LIN {X 0,Y 206.797,Z 825.336,A -85,B 0,C 180,E1 6643.136,E2 6643.136} C_VEL
LIN {X 0,Y 199.995,Z 839.74,A -85,B 0,C 180,E1 6641.339,E2 6641.339} C_VEL
LIN {X 0,Y 192.06,Z 853.457,A -85,B 0,C 180,E1 6639.054,E2 6639.054} C_VEL
LIN {X 0,Y 183.757,Z 865.321,A -85,B 0,C 180,E1 6636.388,E2 6636.388} C_VEL
LIN {X 0,Y 174.878,Z 876.071,A -85,B 0,C 180,E1 6633.098,E2 6633.098} C_VEL
LIN {X 0,Y 165.992,Z 885.275,A -85,B 0,C 180,E1 6629.202,E2 6629.202} C_VEL
LIN {X 0,Y 157.179,Z 892.943,A -85,B 0,C 180,E1 6624.498,E2 6624.498} C_VEL
LIN {X 0,Y 149.304,Z 898.742,A -85,B 0,C 180,E1 6619.164,E2 6619.164} C_VEL
LIN {X 0,Y 142.639,Z 902.668,A -85,B 0,C 180,E1 6613.195,E2 6613.195} C_VEL
LIN {X 0,Y 137.177,Z 904.906,A -85,B 0,C 180,E1 6606.175,E2 6606.175} C_VEL
LIN {X 0,Y 133.759,Z 905.166,A -85,B 0,C 180,E1 6599.061,E2 6599.061} C_VEL
LIN {X 0,Y 132.061,Z 903.501,A -85,B 0,C 180,E1 6591.365,E2 6591.365} C_VEL
LIN {X 0,Y 132.109,Z 900.299,A -85,B 0,C 180,E1 6584.356,E2 6584.356} C_VEL
LIN {X 0,Y 133.672,Z 895.163,A -85,B 0,C 180,E1 6577.3,E2 6577.3} C_VEL
LIN {X 0,Y 136.579,Z 888.49,A -85,B 0,C 180,E1 6570.834,E2 6570.834} C_VEL
LIN {X 0,Y 140.519,Z 880.369,A -85,B 0,C 180,E1 6565.097,E2 6565.097} C_VEL
LIN {X 0,Y 145.58,Z 870.087,A -85,B 0,C 180,E1 6559.71,E2 6559.71} C_VEL
LIN {X 0,Y 150.721,Z 859.162,A -85,B 0,C 180,E1 6555.396,E2 6555.396} C_VEL
LIN {X 0,Y 156.249,Z 846.148,A -85,B 0,C 180,E1 6551.53,E2 6551.53} C_VEL
LIN {X 0,Y 161.502,Z 832.108,A -85,B 0,C 180,E1 6548.383,E2 6548.383} C_VEL
LIN {X 0,Y 166.228,Z 816.841,A -85,B 0,C 180,E1 6545.854,E2 6545.854} C_VEL
LIN {X 0,Y 170.099,Z 801.128,A -85,B 0,C 180,E1 6543.933,E2 6543.933} C_VEL
LIN {X 0,Y 173.031,Z 784.414,A -85,B 0,C 180,E1 6542.51,E2 6542.51} C_VEL
LIN {X 0,Y 174.929,Z 766.861,A -85,B 0,C 180,E1 6541.561,E2 6541.561} C_VEL
LIN {X 0,Y 180.831,Z 690.748,A -85,B 0,C 180,E1 6538.945,E2 6538.945} C_VEL
LIN {X 0,Y 178.846,Z 660.983,A -85,B 0,C 180,E1 6536.338,E2 6536.338} C_VEL
LIN {X 0,Y 173.079,Z 648.188,A -85,B 0,C 180,E1 6533.021,E2 6533.021} C_VEL
LIN {X 0,Y 167.452,Z 637.292,A -85,B 0,C 180,E1 6529.394,E2 6529.394} C_VEL
LIN {X 0,Y 162.798,Z 629.498,A -85,B 0,C 180,E1 6526.02,E2 6526.02} C_VEL
LIN {X 0,Y 160.162,Z 624.669,A -85,B 0,C 180,E1 6523.599,E2 6523.599} C_VEL
LIN {X 0,Y 158.656,Z 618.749,A -85,B 0,C 180,E1 6518.142,E2 6518.142} C_VEL
LIN {X 0,Y 157.464,Z 614.043,A -85,B 0,C 180,E1 6512.666,E2 6512.666} C_VEL
LIN {X 0,Y 156.476,Z 610.789,A -85,B 0,C 180,E1 6507.354,E2 6507.354} C_VEL
LIN {X 0,Y 155.784,Z 607.867,A -85,B 0,C 180,E1 6499.888,E2 6499.888} C_VEL
LIN {X 0,Y 155.499,Z 607.423,A -85,B 0,C 180,E1 6493.007,E2 6493.007} C_VEL
LIN {X 0,Y 156.212,Z 608.246,A -85,B 0,C 180,E1 6486.248,E2 6486.248} C_VEL
LIN {X 0,Y 157.742,Z 612.427,A -85,B 0,C 180,E1 6477.458,E2 6477.458} C_VEL
LIN {X 0,Y 159.064,Z 616.319,A -85,B 0,C 180,E1 6472.415,E2 6472.415} C_VEL
LIN {X 0,Y 160.623,Z 620.813,A -85,B 0,C 180,E1 6467.768,E2 6467.768} C_VEL
LIN {X 0,Y 161.663,Z 623.295,A -85,B 0,C 180,E1 6465.951,E2 6465.951} C_VEL
LIN {X 0,Y 166.617,Z 630.679,A -85,B 0,C 180,E1 6462.27,E2 6462.27} C_VEL
LIN {X 0,Y 171.386,Z 638.352,A -85,B 0,C 180,E1 6459.154,E2 6459.154} C_VEL
LIN {X 0,Y 177.675,Z 649.622,A -85,B 0,C 180,E1 6455.524,E2 6455.524} C_VEL
LIN {X 0,Y 184.39,Z 663.539,A -85,B 0,C 180,E1 6452.072,E2 6452.072} C_VEL
LIN {X 0,Y 186.181,Z 667.991,A -85,B 0,C 180,E1 6451.177,E2 6451.177} C_VEL
LIN {X 0,Y 176.469,Z 794.423,A -85,B 0,C 180,E1 6447.137,E2 6447.137} C_VEL
LIN {X 0,Y 173.768,Z 812.549,A -85,B 0,C 180,E1 6446.085,E2 6446.085} C_VEL
LIN {X 0,Y 169.856,Z 829.853,A -85,B 0,C 180,E1 6444.615,E2 6444.615} C_VEL
LIN {X 0,Y 164.877,Z 846.635,A -85,B 0,C 180,E1 6442.601,E2 6442.601} C_VEL
LIN {X 0,Y 159.263,Z 862.335,A -85,B 0,C 180,E1 6439.99,E2 6439.99} C_VEL
LIN {X 0,Y 153.152,Z 877.3,A -85,B 0,C 180,E1 6436.64,E2 6436.64} C_VEL
LIN {X 0,Y 149.717,Z 883.178,A -85,B 0,C 180,E1 6435.221,E2 6435.221} C_VEL
LIN {X 0,Y 140.413,Z 893.8,A -85,B 0,C 180,E1 6432.527,E2 6432.527} C_VEL
LIN {X 0,Y 135.698,Z 899.523,A -85,B 0,C 180,E1 6430.471,E2 6430.471} C_VEL
LIN {X 0,Y 134.427,Z 901.633,A -85,B 0,C 180,E1 6429.517,E2 6429.517} C_VEL
LIN {X 0,Y 128.939,Z 912.824,A -85,B 0,C 180,E1 6423.409,E2 6423.409} C_VEL
LIN {X 0,Y 124.88,Z 922.114,A -85,B 0,C 180,E1 6416.643,E2 6416.643} C_VEL
LIN {X 0,Y 122.49,Z 929.902,A -85,B 0,C 180,E1 6409.062,E2 6409.062} C_VEL
LIN {X 0,Y 122.057,Z 935.728,A -85,B 0,C 180,E1 6401.343,E2 6401.343} C_VEL
LIN {X 0,Y 123.276,Z 939.721,A -85,B 0,C 180,E1 6393.726,E2 6393.726} C_VEL
LIN {X 0,Y 124.129,Z 941.024,A -85,B 0,C 180,E1 6390.006,E2 6390.006} C_VEL
LIN {X 0,Y 122.525,Z 941.678,A -85,B 0,C 180,E1 6383.917,E2 6383.917} C_VEL
LIN {X 0,Y 121.616,Z 940.962,A -85,B 0,C 180,E1 6375.242,E2 6375.242} C_VEL
LIN {X 0,Y 123.356,Z 938.365,A -85,B 0,C 180,E1 6366.335,E2 6366.335} C_VEL
LIN {X 0,Y 127.941,Z 933.894,A -85,B 0,C 180,E1 6357.908,E2 6357.908} C_VEL
LIN {X 0,Y 135.11,Z 927.559,A -85,B 0,C 180,E1 6350.32,E2 6350.32} C_VEL
LIN {X 0,Y 143.929,Z 919.636,A -85,B 0,C 180,E1 6344.002,E2 6344.002} C_VEL
LIN {X 0,Y 153.262,Z 910.652,A -85,B 0,C 180,E1 6339.087,E2 6339.087} C_VEL
LIN {X 0,Y 163.414,Z 899.916,A -85,B 0,C 180,E1 6334.941,E2 6334.941} C_VEL
LIN {X 0,Y 173.651,Z 887.696,A -85,B 0,C 180,E1 6331.568,E2 6331.568} C_VEL
LIN {X 0,Y 183.343,Z 874.475,A -85,B 0,C 180,E1 6328.938,E2 6328.938} C_VEL
LIN {X 0,Y 192.098,Z 860.475,A -85,B 0,C 180,E1 6326.925,E2 6326.925} C_VEL
LIN {X 0,Y 200.177,Z 845.013,A -85,B 0,C 180,E1 6325.32,E2 6325.32} C_VEL
LIN {X 0,Y 207.015,Z 828.852,A -85,B 0,C 180,E1 6324.118,E2 6324.118} C_VEL
LIN {X 0,Y 212.408,Z 812.263,A -85,B 0,C 180,E1 6323.227,E2 6323.227} C_VEL
LIN {X 0,Y 216.347,Z 794.64,A -85,B 0,C 180,E1 6322.56,E2 6322.56} C_VEL
LIN {X 0,Y 219.19,Z 771.808,A -85,B 0,C 180,E1 6321.967,E2 6321.967} C_VEL
LIN {X 0,Y 226.117,Z 704.464,A -85,B 0,C 180,E1 6320.324,E2 6320.324} C_VEL
LIN {X 0,Y 224.098,Z 700.142,A -85,B 0,C 180,E1 6317.93,E2 6317.93} C_VEL
LIN {X 0,Y 222.421,Z 696.804,A -85,B 0,C 180,E1 6315.513,E2 6315.513} C_VEL
LIN {X 0,Y 220.756,Z 693.625,A -85,B 0,C 180,E1 6312.423,E2 6312.423} C_VEL
LIN {X 0,Y 219.702,Z 691.808,A -85,B 0,C 180,E1 6309.429,E2 6309.429} C_VEL
LIN {X 0,Y 219.018,Z 691.339,A -85,B 0,C 180,E1 6304.451,E2 6304.451} C_VEL
LIN {X 0,Y 219.877,Z 694.271,A -85,B 0,C 180,E1 6299.088,E2 6299.088} C_VEL
LIN {X 0,Y 221.873,Z 699.904,A -85,B 0,C 180,E1 6294.504,E2 6294.504} C_VEL
LIN {X 0,Y 223.806,Z 705.62,A -85,B 0,C 180,E1 6291.457,E2 6291.457} C_VEL
LIN {X 0,Y 224.774,Z 708.661,A -85,B 0,C 180,E1 6290.16,E2 6290.16} C_VEL
LIN {X 0,Y 217.189,Z 777.924,A -85,B 0,C 180,E1 6288.398,E2 6288.398} C_VEL
LIN {X 0,Y 214.061,Z 794.611,A -85,B 0,C 180,E1 6287.636,E2 6287.636} C_VEL
LIN {X 0,Y 209.414,Z 811.1,A -85,B 0,C 180,E1 6286.545,E2 6286.545} C_VEL
LIN {X 0,Y 203.709,Z 826.111,A -85,B 0,C 180,E1 6285.192,E2 6285.192} C_VEL
LIN {X 0,Y 196.776,Z 840.356,A -85,B 0,C 180,E1 6283.468,E2 6283.468} C_VEL
LIN {X 0,Y 188.507,Z 854.189,A -85,B 0,C 180,E1 6281.227,E2 6281.227} C_VEL
LIN {X 0,Y 179.816,Z 866.183,A -85,B 0,C 180,E1 6278.598,E2 6278.598} C_VEL
LIN {X 0,Y 170.497,Z 876.991,A -85,B 0,C 180,E1 6275.343,E2 6275.343} C_VEL
LIN {X 0,Y 161.105,Z 886.255,A -85,B 0,C 180,E1 6271.452,E2 6271.452} C_VEL
LIN {X 0,Y 151.804,Z 893.915,A -85,B 0,C 180,E1 6266.755,E2 6266.755} C_VEL
LIN {X 0,Y 143.37,Z 899.764,A -85,B 0,C 180,E1 6261.346,E2 6261.346} C_VEL
LIN {X 0,Y 136.05,Z 903.81,A -85,B 0,C 180,E1 6255.127,E2 6255.127} C_VEL
LIN {X 0,Y 130.112,Z 906.063,A -85,B 0,C 180,E1 6247.924,E2 6247.924} C_VEL
LIN {X 0,Y 126.249,Z 906.414,A -85,B 0,C 180,E1 6240.446,E2 6240.446} C_VEL
LIN {X 0,Y 124.277,Z 904.937,A -85,B 0,C 180,E1 6232.709,E2 6232.709} C_VEL
LIN {X 0,Y 124.116,Z 901.684,A -85,B 0,C 180,E1 6224.824,E2 6224.824} C_VEL
LIN {X 0,Y 125.65,Z 896.658,A -85,B 0,C 180,E1 6217.309,E2 6217.309} C_VEL
LIN {X 0,Y 128.631,Z 890.083,A -85,B 0,C 180,E1 6210.44,E2 6210.44} C_VEL
LIN {X 0,Y 132.727,Z 882.138,A -85,B 0,C 180,E1 6204.375,E2 6204.375} C_VEL
LIN {X 0,Y 138.002,Z 872.008,A -85,B 0,C 180,E1 6198.715,E2 6198.715} C_VEL
LIN {X 0,Y 143.422,Z 861.174,A -85,B 0,C 180,E1 6194.171,E2 6194.171} C_VEL
LIN {X 0,Y 149.119,Z 848.632,A -85,B 0,C 180,E1 6190.219,E2 6190.219} C_VEL
LIN {X 0,Y 154.882,Z 834.127,A -85,B 0,C 180,E1 6186.807,E2 6186.807} C_VEL
LIN {X 0,Y 159.53,Z 820.265,A -85,B 0,C 180,E1 6184.374,E2 6184.374} C_VEL
LIN {X 0,Y 163.708,Z 804.613,A -85,B 0,C 180,E1 6182.341,E2 6182.341} C_VEL
LIN {X 0,Y 167.041,Z 787.803,A -85,B 0,C 180,E1 6180.787,E2 6180.787} C_VEL
LIN {X 0,Y 169.167,Z 770.445,A -85,B 0,C 180,E1 6179.766,E2 6179.766} C_VEL
LIN {X 0,Y 175.546,Z 691.754,A -85,B 0,C 180,E1 6177.022,E2 6177.022} C_VEL
LIN {X 0,Y 174.014,Z 664.859,A -85,B 0,C 180,E1 6174.603,E2 6174.603} C_VEL
LIN {X 0,Y 169.097,Z 653.532,A -85,B 0,C 180,E1 6171.512,E2 6171.512} C_VEL
LIN {X 0,Y 164.039,Z 643.286,A -85,B 0,C 180,E1 6167.972,E2 6167.972} C_VEL
LIN {X 0,Y 159.863,Z 635.985,A -85,B 0,C 180,E1 6164.72,E2 6164.72} C_VEL
LIN {X 0,Y 156.446,Z 630.229,A -85,B 0,C 180,E1 6161.658,E2 6161.658} C_VEL
LIN {X 0,Y 153.087,Z 624.474,A -85,B 0,C 180,E1 6157.876,E2 6157.876} C_VEL
LIN {X 0,Y 151.949,Z 619.733,A -85,B 0,C 180,E1 6152.209,E2 6152.209} C_VEL
LIN {X 0,Y 151.071,Z 616.555,A -85,B 0,C 180,E1 6146.684,E2 6146.684} C_VEL
LIN {X 0,Y 150.561,Z 613.897,A -85,B 0,C 180,E1 6139.394,E2 6139.394} C_VEL
LIN {X 0,Y 150.388,Z 613.572,A -85,B 0,C 180,E1 6132.285,E2 6132.285} C_VEL
LIN {X 0,Y 151.1,Z 614.41,A -85,B 0,C 180,E1 6126.078,E2 6126.078} C_VEL
LIN {X 0,Y 152.426,Z 618.381,A -85,B 0,C 180,E1 6117.745,E2 6117.745} C_VEL
LIN {X 0,Y 153.595,Z 622.011,A -85,B 0,C 180,E1 6112.896,E2 6112.896} C_VEL
LIN {X 0,Y 155.127,Z 624.627,A -85,B 0,C 180,E1 6110.728,E2 6110.728} C_VEL
LIN {X 0,Y 159.593,Z 631.048,A -85,B 0,C 180,E1 6106.597,E2 6106.597} C_VEL
LIN {X 0,Y 163.835,Z 637.647,A -85,B 0,C 180,E1 6103.278,E2 6103.278} C_VEL
LIN {X 0,Y 169.053,Z 646.383,A -85,B 0,C 180,E1 6099.713,E2 6099.713} C_VEL
LIN {X 0,Y 175.672,Z 659.281,A -85,B 0,C 180,E1 6095.719,E2 6095.719} C_VEL
LIN {X 0,Y 180.73,Z 670.642,A -85,B 0,C 180,E1 6092.985,E2 6092.985} C_VEL
LIN {X 0,Y 170.871,Z 793.82,A -85,B 0,C 180,E1 6089.028,E2 6089.028} C_VEL
LIN {X 0,Y 168.065,Z 811.932,A -85,B 0,C 180,E1 6087.969,E2 6087.969} C_VEL
LIN {X 0,Y 163.998,Z 829.277,A -85,B 0,C 180,E1 6086.485,E2 6086.485} C_VEL
LIN {X 0,Y 159.083,Z 845.278,A -85,B 0,C 180,E1 6084.56,E2 6084.56} C_VEL
LIN {X 0,Y 153.136,Z 861.262,A -85,B 0,C 180,E1 6081.886,E2 6081.886} C_VEL
LIN {X 0,Y 146.523,Z 876.72,A -85,B 0,C 180,E1 6078.352,E2 6078.352} C_VEL
LIN {X 0,Y 140.034,Z 890.42,A -85,B 0,C 180,E1 6074.122,E2 6074.122} C_VEL
LIN {X 0,Y 134.427,Z 901.633,A -85,B 0,C 180,E1 6069.517,E2 6069.517} C_VEL
LIN {X 0,Y 131.1,Z 906.417,A -85,B 0,C 180,E1 6067.262,E2 6067.262} C_VEL
LIN {X 0,Y 121.766,Z 915.195,A -85,B 0,C 180,E1 6062.347,E2 6062.347} C_VEL
LIN {X 0,Y 117.995,Z 919.49,A -85,B 0,C 180,E1 6059.091,E2 6059.091} C_VEL
LIN {X 0,Y 117.439,Z 920.53,A -85,B 0,C 180,E1 6058.18,E2 6058.18} C_VEL
LIN {X 0,Y 114.755,Z 928.174,A -85,B 0,C 180,E1 6050.401,E2 6050.401} C_VEL
LIN {X 0,Y 114.071,Z 934.162,A -85,B 0,C 180,E1 6042.149,E2 6042.149} C_VEL
LIN {X 0,Y 115.254,Z 938.342,A -85,B 0,C 180,E1 6033.936,E2 6033.936} C_VEL
LIN {X 0,Y 116.116,Z 939.794,A -85,B 0,C 180,E1 6029.513,E2 6029.513} C_VEL
LIN {X 0,Y 114.102,Z 940.429,A -85,B 0,C 180,E1 6021.44,E2 6021.44} C_VEL
LIN {X 0,Y 113.938,Z 939.373,A -85,B 0,C 180,E1 6012.121,E2 6012.121} C_VEL
LIN {X 0,Y 116.855,Z 936.376,A -85,B 0,C 180,E1 6002.49,E2 6002.49} C_VEL
LIN {X 0,Y 122.547,Z 931.741,A -85,B 0,C 180,E1 5994.035,E2 5994.035} C_VEL
LIN {X 0,Y 130.766,Z 925.204,A -85,B 0,C 180,E1 5986.528,E2 5986.528} C_VEL
LIN {X 0,Y 140.569,Z 916.932,A -85,B 0,C 180,E1 5980.336,E2 5980.336} C_VEL
LIN {X 0,Y 151,Z 907.368,A -85,B 0,C 180,E1 5975.481,E2 5975.481} C_VEL
LIN {X 0,Y 161.874,Z 896.237,A -85,B 0,C 180,E1 5971.543,E2 5971.543} C_VEL
LIN {X 0,Y 172.318,Z 883.95,A -85,B 0,C 180,E1 5968.488,E2 5968.488} C_VEL
LIN {X 0,Y 182.466,Z 870.071,A -85,B 0,C 180,E1 5966.035,E2 5966.035} C_VEL
LIN {X 0,Y 191.297,Z 855.826,A -85,B 0,C 180,E1 5964.227,E2 5964.227} C_VEL
LIN {X 0,Y 199.209,Z 840.45,A -85,B 0,C 180,E1 5962.824,E2 5962.824} C_VEL
LIN {X 0,Y 205.646,Z 824.728,A -85,B 0,C 180,E1 5961.797,E2 5961.797} C_VEL
LIN {X 0,Y 210.965,Z 807.432,A -85,B 0,C 180,E1 5960.984,E2 5960.984} C_VEL
LIN {X 0,Y 214.67,Z 789.539,A -85,B 0,C 180,E1 5960.387,E2 5960.387} C_VEL
LIN {X 0,Y 223.44,Z 709.576,A -85,B 0,C 180,E1 5958.524,E2 5958.524} C_VEL
LIN {X 0,Y 221.157,Z 704.655,A -85,B 0,C 180,E1 5955.201,E2 5955.201} C_VEL
LIN {X 0,Y 219.506,Z 701.33,A -85,B 0,C 180,E1 5951.961,E2 5951.961} C_VEL
LIN {X 0,Y 218.618,Z 699.699,A -85,B 0,C 180,E1 5949.211,E2 5949.211} C_VEL
LIN {X 0,Y 217.994,Z 699.283,A -85,B 0,C 180,E1 5944.472,E2 5944.472} C_VEL
LIN {X 0,Y 218.746,Z 702.191,A -85,B 0,C 180,E1 5939.345,E2 5939.345} C_VEL
LIN {X 0,Y 220.421,Z 707.445,A -85,B 0,C 180,E1 5935.12,E2 5935.12} C_VEL
LIN {X 0,Y 222.09,Z 712.85,A -85,B 0,C 180,E1 5932.237,E2 5932.237} C_VEL
LIN {X 0,Y 222.179,Z 713.622,A -85,B 0,C 180,E1 5932.033,E2 5932.033} C_VEL
LIN {X 0,Y 214.798,Z 778.829,A -85,B 0,C 180,E1 5930.41,E2 5930.41} C_VEL
LIN {X 0,Y 211.524,Z 795.574,A -85,B 0,C 180,E1 5929.663,E2 5929.663} C_VEL
LIN {X 0,Y 206.647,Z 812.229,A -85,B 0,C 180,E1 5928.589,E2 5928.589} C_VEL
LIN {X 0,Y 200.857,Z 826.96,A -85,B 0,C 180,E1 5927.3,E2 5927.3} C_VEL
LIN {X 0,Y 193.534,Z 841.508,A -85,B 0,C 180,E1 5925.591,E2 5925.591} C_VEL
LIN {X 0,Y 185.253,Z 854.896,A -85,B 0,C 180,E1 5923.485,E2 5923.485} C_VEL
LIN {X 0,Y 176.183,Z 867.013,A -85,B 0,C 180,E1 5920.912,E2 5920.912} C_VEL
LIN {X 0,Y 166.394,Z 877.92,A -85,B 0,C 180,E1 5917.703,E2 5917.703} C_VEL
LIN {X 0,Y 156.498,Z 887.247,A -85,B 0,C 180,E1 5913.842,E2 5913.842} C_VEL
LIN {X 0,Y 146.972,Z 894.728,A -85,B 0,C 180,E1 5909.32,E2 5909.32} C_VEL
LIN {X 0,Y 137.664,Z 900.802,A -85,B 0,C 180,E1 5903.711,E2 5903.711} C_VEL
LIN {X 0,Y 129.988,Z 904.81,A -85,B 0,C 180,E1 5897.584,E2 5897.584} C_VEL
LIN {X 0,Y 123.522,Z 907.134,A -85,B 0,C 180,E1 5890.347,E2 5890.347} C_VEL
LIN {X 0,Y 119.031,Z 907.663,A -85,B 0,C 180,E1 5882.51,E2 5882.51} C_VEL
LIN {X 0,Y 116.575,Z 906.395,A -85,B 0,C 180,E1 5874.302,E2 5874.302} C_VEL
LIN {X 0,Y 116.085,Z 903.355,A -85,B 0,C 180,E1 5865.991,E2 5865.991} C_VEL
LIN {X 0,Y 117.48,Z 898.534,A -85,B 0,C 180,E1 5857.82,E2 5857.82} C_VEL
LIN {X 0,Y 120.437,Z 892.16,A -85,B 0,C 180,E1 5850.47,E2 5850.47} C_VEL
LIN {X 0,Y 124.953,Z 883.846,A -85,B 0,C 180,E1 5843.563,E2 5843.563} C_VEL
LIN {X 0,Y 130.036,Z 874.712,A -85,B 0,C 180,E1 5838.013,E2 5838.013} C_VEL
LIN {X 0,Y 136.07,Z 863.355,A -85,B 0,C 180,E1 5832.903,E2 5832.903} C_VEL
LIN {X 0,Y 142.106,Z 850.977,A -85,B 0,C 180,E1 5828.752,E2 5828.752} C_VEL
LIN {X 0,Y 147.794,Z 837.58,A -85,B 0,C 180,E1 5825.411,E2 5825.411} C_VEL
LIN {X 0,Y 153.242,Z 822.502,A -85,B 0,C 180,E1 5822.611,E2 5822.611} C_VEL
LIN {X 0,Y 157.607,Z 807.353,A -85,B 0,C 180,E1 5820.548,E2 5820.548} C_VEL
LIN {X 0,Y 161.329,Z 789.955,A -85,B 0,C 180,E1 5818.872,E2 5818.872} C_VEL
LIN {X 0,Y 163.632,Z 773.206,A -85,B 0,C 180,E1 5817.82,E2 5817.82} C_VEL
LIN {X 0,Y 170.445,Z 692.643,A -85,B 0,C 180,E1 5814.976,E2 5814.976} C_VEL
LIN {X 0,Y 169.238,Z 668.376,A -85,B 0,C 180,E1 5812.691,E2 5812.691} C_VEL
LIN {X 0,Y 164.545,Z 657.344,A -85,B 0,C 180,E1 5809.427,E2 5809.427} C_VEL
LIN {X 0,Y 160.242,Z 648.452,A -85,B 0,C 180,E1 5806.138,E2 5806.138} C_VEL
LIN {X 0,Y 156.778,Z 642.053,A -85,B 0,C 180,E1 5803.158,E2 5803.158} C_VEL
LIN {X 0,Y 153.945,Z 637.012,A -85,B 0,C 180,E1 5800.382,E2 5800.382} C_VEL
LIN {X 0,Y 150.483,Z 631.184,A -85,B 0,C 180,E1 5796.414,E2 5796.414} C_VEL
LIN {X 0,Y 146.365,Z 624.737,A -85,B 0,C 180,E1 5790.14,E2 5790.14} C_VEL
LIN {X 0,Y 145.777,Z 622.529,A -85,B 0,C 180,E1 5786.477,E2 5786.477} C_VEL
LIN {X 0,Y 145.38,Z 619.986,A -85,B 0,C 180,E1 5779.277,E2 5779.277} C_VEL
LIN {X 0,Y 145.254,Z 619.707,A -85,B 0,C 180,E1 5772.188,E2 5772.188} C_VEL
LIN {X 0,Y 145.95,Z 620.629,A -85,B 0,C 180,E1 5765.899,E2 5765.899} C_VEL
LIN {X 0,Y 146.979,Z 623.577,A -85,B 0,C 180,E1 5759.81,E2 5759.81} C_VEL
LIN {X 0,Y 151.536,Z 629.748,A -85,B 0,C 180,E1 5753.37,E2 5753.37} C_VEL
LIN {X 0,Y 156.619,Z 637.264,A -85,B 0,C 180,E1 5748.119,E2 5748.119} C_VEL
LIN {X 0,Y 160.878,Z 644.227,A -85,B 0,C 180,E1 5744.5,E2 5744.5} C_VEL
LIN {X 0,Y 165.92,Z 653.119,A -85,B 0,C 180,E1 5740.827,E2 5740.827} C_VEL
LIN {X 0,Y 171.873,Z 665.286,A -85,B 0,C 180,E1 5736.97,E2 5736.97} C_VEL
LIN {X 0,Y 175.395,Z 673.677,A -85,B 0,C 180,E1 5734.882,E2 5734.882} C_VEL
LIN {X 0,Y 165.404,Z 793.304,A -85,B 0,C 180,E1 5731.023,E2 5731.023} C_VEL
LIN {X 0,Y 162.47,Z 811.512,A -85,B 0,C 180,E1 5729.953,E2 5729.953} C_VEL
LIN {X 0,Y 158.326,Z 828.545,A -85,B 0,C 180,E1 5728.491,E2 5728.491} C_VEL
LIN {X 0,Y 153.312,Z 844.305,A -85,B 0,C 180,E1 5726.593,E2 5726.593} C_VEL
LIN {X 0,Y 147.191,Z 860.137,A -85,B 0,C 180,E1 5723.937,E2 5723.937} C_VEL
LIN {X 0,Y 140.255,Z 875.651,A -85,B 0,C 180,E1 5720.348,E2 5720.348} C_VEL
LIN {X 0,Y 133.413,Z 889.39,A -85,B 0,C 180,E1 5716.013,E2 5716.013} C_VEL
LIN {X 0,Y 126.987,Z 901.471,A -85,B 0,C 180,E1 5710.81,E2 5710.81} C_VEL
LIN {X 0,Y 121.313,Z 912.331,A -85,B 0,C 180,E1 5704.494,E2 5704.494} C_VEL
LIN {X 0,Y 117.439,Z 920.53,A -85,B 0,C 180,E1 5698.18,E2 5698.18} C_VEL
LIN {X 0,Y 115.059,Z 923.981,A -85,B 0,C 180,E1 5694.949,E2 5694.949} C_VEL
LIN {X 0,Y 109.226,Z 928.964,A -85,B 0,C 180,E1 5688.951,E2 5688.951} C_VEL
LIN {X 0,Y 106.375,Z 932.005,A -85,B 0,C 180,E1 5684.086,E2 5684.086} C_VEL
LIN {X 0,Y 106.127,Z 933.171,A -85,B 0,C 180,E1 5682.088,E2 5682.088} C_VEL
LIN {X 0,Y 107.446,Z 937.297,A -85,B 0,C 180,E1 5673.207,E2 5673.207} C_VEL
LIN {X 0,Y 108.142,Z 938.461,A -85,B 0,C 180,E1 5669.477,E2 5669.477} C_VEL
LIN {X 0,Y 106.079,Z 939.156,A -85,B 0,C 180,E1 5660.787,E2 5660.787} C_VEL
LIN {X 0,Y 106.173,Z 938.215,A -85,B 0,C 180,E1 5650.764,E2 5650.764} C_VEL
LIN {X 0,Y 109.628,Z 935.314,A -85,B 0,C 180,E1 5640.505,E2 5640.505} C_VEL
LIN {X 0,Y 115.992,Z 930.774,A -85,B 0,C 180,E1 5631.649,E2 5631.649} C_VEL
LIN {X 0,Y 124.933,Z 924.362,A -85,B 0,C 180,E1 5623.935,E2 5623.935} C_VEL
LIN {X 0,Y 135.29,Z 916.317,A -85,B 0,C 180,E1 5617.756,E2 5617.756} C_VEL
LIN {X 0,Y 146.419,Z 906.787,A -85,B 0,C 180,E1 5612.883,E2 5612.883} C_VEL
LIN {X 0,Y 157.777,Z 895.773,A -85,B 0,C 180,E1 5609.029,E2 5609.029} C_VEL
LIN {X 0,Y 168.613,Z 883.672,A -85,B 0,C 180,E1 5606.074,E2 5606.074} C_VEL
LIN {X 0,Y 179.079,Z 869.937,A -85,B 0,C 180,E1 5603.72,E2 5603.72} C_VEL
LIN {X 0,Y 188.584,Z 855.121,A -85,B 0,C 180,E1 5601.922,E2 5601.922} C_VEL
LIN {X 0,Y 196.542,Z 840.095,A -85,B 0,C 180,E1 5600.625,E2 5600.625} C_VEL
LIN {X 0,Y 203.454,Z 823.627,A -85,B 0,C 180,E1 5599.613,E2 5599.613} C_VEL
LIN {X 0,Y 208.924,Z 806.135,A -85,B 0,C 180,E1 5598.846,E2 5598.846} C_VEL
LIN {X 0,Y 212.648,Z 788.413,A -85,B 0,C 180,E1 5598.291,E2 5598.291} C_VEL
LIN {X 0,Y 220.962,Z 714.999,A -85,B 0,C 180,E1 5596.631,E2 5596.631} C_VEL
LIN {X 0,Y 219.463,Z 711.628,A -85,B 0,C 180,E1 5594.107,E2 5594.107} C_VEL
LIN {X 0,Y 218.147,Z 708.747,A -85,B 0,C 180,E1 5591.098,E2 5591.098} C_VEL
LIN {X 0,Y 217.471,Z 707.525,A -85,B 0,C 180,E1 5588.726,E2 5588.726} C_VEL
LIN {X 0,Y 216.967,Z 707.251,A -85,B 0,C 180,E1 5584.493,E2 5584.493} C_VEL
LIN {X 0,Y 217.589,Z 709.978,A -85,B 0,C 180,E1 5579.736,E2 5579.736} C_VEL
LIN {X 0,Y 218.995,Z 714.983,A -85,B 0,C 180,E1 5575.745,E2 5575.745} C_VEL
LIN {X 0,Y 219.876,Z 718.315,A -85,B 0,C 180,E1 5573.956,E2 5573.956} C_VEL
LIN {X 0,Y 212.716,Z 779.777,A -85,B 0,C 180,E1 5572.466,E2 5572.466} C_VEL
LIN {X 0,Y 209.284,Z 796.659,A -85,B 0,C 180,E1 5571.734,E2 5571.734} C_VEL
LIN {X 0,Y 204.282,Z 813.194,A -85,B 0,C 180,E1 5570.704,E2 5570.704} C_VEL
LIN {X 0,Y 198.288,Z 827.925,A -85,B 0,C 180,E1 5569.461,E2 5569.461} C_VEL
LIN {X 0,Y 190.74,Z 842.424,A -85,B 0,C 180,E1 5567.819,E2 5567.819} C_VEL
LIN {X 0,Y 182.001,Z 856.046,A -85,B 0,C 180,E1 5565.745,E2 5565.745} C_VEL
LIN {X 0,Y 172.854,Z 867.838,A -85,B 0,C 180,E1 5563.319,E2 5563.319} C_VEL
LIN {X 0,Y 162.587,Z 878.847,A -85,B 0,C 180,E1 5560.177,E2 5560.177} C_VEL
LIN {X 0,Y 152.185,Z 888.232,A -85,B 0,C 180,E1 5556.373,E2 5556.373} C_VEL
LIN {X 0,Y 142.084,Z 895.786,A -85,B 0,C 180,E1 5551.868,E2 5551.868} C_VEL
LIN {X 0,Y 132.217,Z 901.852,A -85,B 0,C 180,E1 5546.272,E2 5546.272} C_VEL
LIN {X 0,Y 123.911,Z 905.917,A -85,B 0,C 180,E1 5540.032,E2 5540.032} C_VEL
LIN {X 0,Y 116.794,Z 908.298,A -85,B 0,C 180,E1 5532.543,E2 5532.543} C_VEL
LIN {X 0,Y 111.73,Z 908.88,A -85,B 0,C 180,E1 5524.307,E2 5524.307} C_VEL
LIN {X 0,Y 108.851,Z 907.707,A -85,B 0,C 180,E1 5515.567,E2 5515.567} C_VEL
LIN {X 0,Y 108.118,Z 904.731,A -85,B 0,C 180,E1 5506.651,E2 5506.651} C_VEL
LIN {X 0,Y 109.447,Z 899.996,A -85,B 0,C 180,E1 5497.869,E2 5497.869} C_VEL
LIN {X 0,Y 112.493,Z 893.746,A -85,B 0,C 180,E1 5489.994,E2 5489.994} C_VEL
LIN {X 0,Y 117.204,Z 885.541,A -85,B 0,C 180,E1 5482.643,E2 5482.643} C_VEL
LIN {X 0,Y 122.535,Z 876.585,A -85,B 0,C 180,E1 5476.788,E2 5476.788} C_VEL
LIN {X 0,Y 128.857,Z 865.421,A -85,B 0,C 180,E1 5471.446,E2 5471.446} C_VEL
LIN {X 0,Y 135.459,Z 852.687,A -85,B 0,C 180,E1 5466.967,E2 5466.967} C_VEL
LIN {X 0,Y 141.42,Z 839.524,A -85,B 0,C 180,E1 5463.547,E2 5463.547} C_VEL
LIN {X 0,Y 147.11,Z 824.682,A -85,B 0,C 180,E1 5460.699,E2 5460.699} C_VEL
LIN {X 0,Y 152.003,Z 808.806,A -85,B 0,C 180,E1 5458.468,E2 5458.468} C_VEL
LIN {X 0,Y 155.872,Z 791.753,A -85,B 0,C 180,E1 5456.792,E2 5456.792} C_VEL
LIN {X 0,Y 158.417,Z 774.779,A -85,B 0,C 180,E1 5455.686,E2 5455.686} C_VEL
LIN {X 0,Y 165.578,Z 693.622,A -85,B 0,C 180,E1 5452.816,E2 5452.816} C_VEL
LIN {X 0,Y 164.709,Z 672.133,A -85,B 0,C 180,E1 5450.715,E2 5450.715} C_VEL
LIN {X 0,Y 160.01,Z 660.662,A -85,B 0,C 180,E1 5447.098,E2 5447.098} C_VEL
LIN {X 0,Y 155.449,Z 651.051,A -85,B 0,C 180,E1 5443.112,E2 5443.112} C_VEL
LIN {X 0,Y 151.523,Z 643.791,A -85,B 0,C 180,E1 5439.064,E2 5439.064} C_VEL
LIN {X 0,Y 148.388,Z 638.241,A -85,B 0,C 180,E1 5435.179,E2 5435.179} C_VEL
LIN {X 0,Y 144.737,Z 632.164,A -85,B 0,C 180,E1 5429.146,E2 5429.146} C_VEL
LIN {X 0,Y 143.245,Z 629.91,A -85,B 0,C 180,E1 5425.644,E2 5425.644} C_VEL
LIN {X 0,Y 141.639,Z 627.034,A -85,B 0,C 180,E1 5418.927,E2 5418.927} C_VEL
LIN {X 0,Y 141.66,Z 626.856,A -85,B 0,C 180,E1 5411.812,E2 5411.812} C_VEL
LIN {X 0,Y 143.108,Z 628.24,A -85,B 0,C 180,E1 5405.815,E2 5405.815} C_VEL
LIN {X 0,Y 146.153,Z 632.151,A -85,B 0,C 180,E1 5399.315,E2 5399.315} C_VEL
LIN {X 0,Y 150.114,Z 637.899,A -85,B 0,C 180,E1 5393.691,E2 5393.691} C_VEL
LIN {X 0,Y 154.371,Z 644.556,A -85,B 0,C 180,E1 5389.08,E2 5389.08} C_VEL
LIN {X 0,Y 158.456,Z 651.612,A -85,B 0,C 180,E1 5385.381,E2 5385.381} C_VEL
LIN {X 0,Y 163.644,Z 661.468,A -85,B 0,C 180,E1 5381.383,E2 5381.383} C_VEL
LIN {X 0,Y 169.212,Z 673.708,A -85,B 0,C 180,E1 5377.597,E2 5377.597} C_VEL
LIN {X 0,Y 170.258,Z 676.785,A -85,B 0,C 180,E1 5376.893,E2 5376.893} C_VEL
LIN {X 0,Y 160.173,Z 792.602,A -85,B 0,C 180,E1 5373.16,E2 5373.16} C_VEL
LIN {X 0,Y 157.13,Z 810.818,A -85,B 0,C 180,E1 5372.092,E2 5372.092} C_VEL
LIN {X 0,Y 152.721,Z 828.261,A -85,B 0,C 180,E1 5370.593,E2 5370.593} C_VEL
LIN {X 0,Y 147.478,Z 844.001,A -85,B 0,C 180,E1 5368.677,E2 5368.677} C_VEL
LIN {X 0,Y 141.109,Z 859.72,A -85,B 0,C 180,E1 5366.001,E2 5366.001} C_VEL
LIN {X 0,Y 134.174,Z 874.506,A -85,B 0,C 180,E1 5362.528,E2 5362.528} C_VEL
LIN {X 0,Y 126.954,Z 888.281,A -85,B 0,C 180,E1 5358.098,E2 5358.098} C_VEL
LIN {X 0,Y 119.88,Z 900.81,A -85,B 0,C 180,E1 5352.503,E2 5352.503} C_VEL
LIN {X 0,Y 113.587,Z 912.101,A -85,B 0,C 180,E1 5345.523,E2 5345.523} C_VEL
LIN {X 0,Y 109.102,Z 921.13,A -85,B 0,C 180,E1 5337.869,E2 5337.869} C_VEL
LIN {X 0,Y 106.537,Z 928.58,A -85,B 0,C 180,E1 5329.182,E2 5329.182} C_VEL
LIN {X 0,Y 106.127,Z 933.171,A -85,B 0,C 180,E1 5322.088,E2 5322.088} C_VEL
LIN {X 0,Y 105.434,Z 934.7,A -85,B 0,C 180,E1 5319.007,E2 5319.007} C_VEL
LIN {X 0,Y 102.688,Z 936.139,A -85,B 0,C 180,E1 5314.313,E2 5314.313} C_VEL
LIN {X 0,Y 100.129,Z 937.103,A -85,B 0,C 180,E1 5309.331,E2 5309.331} C_VEL
LIN {X 0,Y 98.003,Z 937.866,A -85,B 0,C 180,E1 5299.426,E2 5299.426} C_VEL
LIN {X 0,Y 98.594,Z 936.94,A -85,B 0,C 180,E1 5288.597,E2 5288.597} C_VEL
LIN {X 0,Y 102.868,Z 934.045,A -85,B 0,C 180,E1 5277.695,E2 5277.695} C_VEL
LIN {X 0,Y 110.626,Z 929.213,A -85,B 0,C 180,E1 5268.036,E2 5268.036} C_VEL
LIN {X 0,Y 119.986,Z 923.115,A -85,B 0,C 180,E1 5260.699,E2 5260.699} C_VEL
LIN {X 0,Y 131.138,Z 915.087,A -85,B 0,C 180,E1 5254.586,E2 5254.586} C_VEL
LIN {X 0,Y 142.927,Z 905.55,A -85,B 0,C 180,E1 5249.854,E2 5249.854} C_VEL
LIN {X 0,Y 154.815,Z 894.515,A -85,B 0,C 180,E1 5246.16,E2 5246.16} C_VEL
LIN {X 0,Y 166.069,Z 882.367,A -85,B 0,C 180,E1 5243.363,E2 5243.363} C_VEL
LIN {X 0,Y 176.433,Z 869.19,A -85,B 0,C 180,E1 5241.238,E2 5241.238} C_VEL
LIN {X 0,Y 186.314,Z 854.256,A -85,B 0,C 180,E1 5239.535,E2 5239.535} C_VEL
LIN {X 0,Y 194.782,Z 838.636,A -85,B 0,C 180,E1 5238.287,E2 5238.287} C_VEL
LIN {X 0,Y 201.649,Z 822.504,A -85,B 0,C 180,E1 5237.379,E2 5237.379} C_VEL
LIN {X 0,Y 207.231,Z 804.874,A -85,B 0,C 180,E1 5236.666,E2 5236.666} C_VEL
LIN {X 0,Y 210.987,Z 787.135,A -85,B 0,C 180,E1 5236.151,E2 5236.151} C_VEL
LIN {X 0,Y 218.72,Z 720.509,A -85,B 0,C 180,E1 5234.697,E2 5234.697} C_VEL
LIN {X 0,Y 217.123,Z 716.85,A -85,B 0,C 180,E1 5231.151,E2 5231.151} C_VEL
LIN {X 0,Y 216.396,Z 715.418,A -85,B 0,C 180,E1 5228.502,E2 5228.502} C_VEL
LIN {X 0,Y 215.937,Z 715.236,A -85,B 0,C 180,E1 5224.514,E2 5224.514} C_VEL
LIN {X 0,Y 216.442,Z 717.764,A -85,B 0,C 180,E1 5220.132,E2 5220.132} C_VEL
LIN {X 0,Y 217.567,Z 722.405,A -85,B 0,C 180,E1 5216.442,E2 5216.442} C_VEL
LIN {X 0,Y 217.767,Z 723.489,A -85,B 0,C 180,E1 5215.907,E2 5215.907} C_VEL
LIN {X 0,Y 210.939,Z 780.557,A -85,B 0,C 180,E1 5214.565,E2 5214.565} C_VEL
LIN {X 0,Y 207.395,Z 797.476,A -85,B 0,C 180,E1 5213.86,E2 5213.86} C_VEL
LIN {X 0,Y 202.407,Z 813.577,A -85,B 0,C 180,E1 5212.905,E2 5212.905} C_VEL
LIN {X 0,Y 196.009,Z 828.922,A -85,B 0,C 180,E1 5211.674,E2 5211.674} C_VEL
LIN {X 0,Y 188.245,Z 843.401,A -85,B 0,C 180,E1 5210.105,E2 5210.105} C_VEL
LIN {X 0,Y 179.034,Z 857.299,A -85,B 0,C 180,E1 5208.074,E2 5208.074} C_VEL
LIN {X 0,Y 169.229,Z 869.393,A -85,B 0,C 180,E1 5205.651,E2 5205.651} C_VEL
LIN {X 0,Y 159.101,Z 879.799,A -85,B 0,C 180,E1 5202.76,E2 5202.76} C_VEL
LIN {X 0,Y 148.188,Z 889.214,A -85,B 0,C 180,E1 5199.046,E2 5199.046} C_VEL
LIN {X 0,Y 137.502,Z 896.84,A -85,B 0,C 180,E1 5194.593,E2 5194.593} C_VEL
LIN {X 0,Y 127.059,Z 902.902,A -85,B 0,C 180,E1 5189.046,E2 5189.046} C_VEL
LIN {X 0,Y 118.085,Z 907.012,A -85,B 0,C 180,E1 5182.726,E2 5182.726} C_VEL
LIN {X 0,Y 110.226,Z 909.472,A -85,B 0,C 180,E1 5174.963,E2 5174.963} C_VEL
LIN {X 0,Y 104.275,Z 910.089,A -85,B 0,C 180,E1 5165.785,E2 5165.785} C_VEL
LIN {X 0,Y 101.05,Z 908.863,A -85,B 0,C 180,E1 5156.43,E2 5156.43} C_VEL
LIN {X 0,Y 100.179,Z 905.784,A -85,B 0,C 180,E1 5146.631,E2 5146.631} C_VEL
LIN {X 0,Y 101.565,Z 901.103,A -85,B 0,C 180,E1 5137.345,E2 5137.345} C_VEL
LIN {X 0,Y 104.83,Z 894.836,A -85,B 0,C 180,E1 5128.9,E2 5128.9} C_VEL
LIN {X 0,Y 109.881,Z 886.627,A -85,B 0,C 180,E1 5121.095,E2 5121.095} C_VEL
LIN {X 0,Y 116.053,Z 876.894,A -85,B 0,C 180,E1 5114.504,E2 5114.504} C_VEL
LIN {X 0,Y 122.841,Z 865.559,A -85,B 0,C 180,E1 5109.01,E2 5109.01} C_VEL
LIN {X 0,Y 129.536,Z 853.295,A -85,B 0,C 180,E1 5104.655,E2 5104.655} C_VEL
LIN {X 0,Y 135.722,Z 840.271,A -85,B 0,C 180,E1 5101.245,E2 5101.245} C_VEL
LIN {X 0,Y 141.832,Z 825.026,A -85,B 0,C 180,E1 5098.316,E2 5098.316} C_VEL
LIN {X 0,Y 146.614,Z 810.244,A -85,B 0,C 180,E1 5096.231,E2 5096.231} C_VEL
LIN {X 0,Y 150.678,Z 793.337,A -85,B 0,C 180,E1 5094.547,E2 5094.547} C_VEL
LIN {X 0,Y 153.474,Z 775.928,A -85,B 0,C 180,E1 5093.392,E2 5093.392} C_VEL
LIN {X 0,Y 160.961,Z 694.634,A -85,B 0,C 180,E1 5090.531,E2 5090.531} C_VEL
LIN {X 0,Y 160.367,Z 675.944,A -85,B 0,C 180,E1 5088.643,E2 5088.643} C_VEL
LIN {X 0,Y 156.243,Z 665.549,A -85,B 0,C 180,E1 5085.133,E2 5085.133} C_VEL
LIN {X 0,Y 152.396,Z 656.961,A -85,B 0,C 180,E1 5081.378,E2 5081.378} C_VEL
LIN {X 0,Y 149.083,Z 650.423,A -85,B 0,C 180,E1 5077.613,E2 5077.613} C_VEL
LIN {X 0,Y 146.32,Z 645.22,A -85,B 0,C 180,E1 5073.844,E2 5073.844} C_VEL
LIN {X 0,Y 143.207,Z 639.596,A -85,B 0,C 180,E1 5068.118,E2 5068.118} C_VEL
LIN {X 0,Y 141.835,Z 637.466,A -85,B 0,C 180,E1 5064.578,E2 5064.578} C_VEL
LIN {X 0,Y 140.607,Z 634.945,A -85,B 0,C 180,E1 5058.664,E2 5058.664} C_VEL
LIN {X 0,Y 140.724,Z 634.844,A -85,B 0,C 180,E1 5051.333,E2 5051.333} C_VEL
LIN {X 0,Y 141.996,Z 636.193,A -85,B 0,C 180,E1 5046.064,E2 5046.064} C_VEL
LIN {X 0,Y 144.636,Z 639.784,A -85,B 0,C 180,E1 5040.1,E2 5040.1} C_VEL
LIN {X 0,Y 148.181,Z 645.236,A -85,B 0,C 180,E1 5034.677,E2 5034.677} C_VEL
LIN {X 0,Y 152,Z 651.538,A -85,B 0,C 180,E1 5030.249,E2 5030.249} C_VEL
LIN {X 0,Y 155.974,Z 658.83,A -85,B 0,C 180,E1 5026.375,E2 5026.375} C_VEL
LIN {X 0,Y 160.684,Z 668.376,A -85,B 0,C 180,E1 5022.482,E2 5022.482} C_VEL
LIN {X 0,Y 165.374,Z 679.494,A -85,B 0,C 180,E1 5019.039,E2 5019.039} C_VEL
LIN {X 0,Y 155.154,Z 792.073,A -85,B 0,C 180,E1 5015.429,E2 5015.429} C_VEL
LIN {X 0,Y 151.999,Z 810.233,A -85,B 0,C 180,E1 5014.37,E2 5014.37} C_VEL
LIN {X 0,Y 147.436,Z 827.638,A -85,B 0,C 180,E1 5012.886,E2 5012.886} C_VEL
LIN {X 0,Y 141.656,Z 844.177,A -85,B 0,C 180,E1 5010.856,E2 5010.856} C_VEL
LIN {X 0,Y 134.986,Z 859.822,A -85,B 0,C 180,E1 5008.141,E2 5008.141} C_VEL
LIN {X 0,Y 127.642,Z 874.646,A -85,B 0,C 180,E1 5004.557,E2 5004.557} C_VEL
LIN {X 0,Y 120.53,Z 887.433,A -85,B 0,C 180,E1 5000.302,E2 5000.302} C_VEL
LIN {X 0,Y 113.401,Z 899.305,A -85,B 0,C 180,E1 4994.862,E2 4994.862} C_VEL
LIN {X 0,Y 106.97,Z 909.986,A -85,B 0,C 180,E1 4988.095,E2 4988.095} C_VEL
LIN {X 0,Y 101.89,Z 919.205,A -85,B 0,C 180,E1 4980.036,E2 4980.036} C_VEL
LIN {X 0,Y 98.811,Z 926.895,A -85,B 0,C 180,E1 4970.748,E2 4970.748} C_VEL
LIN {X 0,Y 98.232,Z 932.575,A -85,B 0,C 180,E1 4961.157,E2 4961.157} C_VEL
LIN {X 0,Y 99.816,Z 936.435,A -85,B 0,C 180,E1 4951.729,E2 4951.729} C_VEL
LIN {X 0,Y 100.161,Z 937.083,A -85,B 0,C 180,E1 4949.435,E2 4949.435} C_VEL
LIN {X 0,Y 100.129,Z 937.103,A -85,B 0,C 180,E1 4949.331,E2 4949.331} C_VEL
LIN {X 0,Y 98.165,Z 937.563,A -85,B 0,C 180,E1 4945.339,E2 4945.339} C_VEL
LIN {X 0,Y 93.679,Z 937.286,A -85,B 0,C 180,E1 4938.848,E2 4938.848} C_VEL
LIN {X 0,Y 90.583,Z 936.395,A -85,B 0,C 180,E1 4931.768,E2 4931.768} C_VEL
LIN {X 0,Y 90.606,Z 935.976,A -85,B 0,C 180,E1 4928.59,E2 4928.59} C_VEL
LIN {X 0,Y 94.969,Z 933.558,A -85,B 0,C 180,E1 4916.819,E2 4916.819} C_VEL
LIN {X 0,Y 102.609,Z 929.431,A -85,B 0,C 180,E1 4906.954,E2 4906.954} C_VEL
LIN {X 0,Y 112.873,Z 923.449,A -85,B 0,C 180,E1 4898.799,E2 4898.799} C_VEL
LIN {X 0,Y 124.472,Z 915.918,A -85,B 0,C 180,E1 4892.513,E2 4892.513} C_VEL
LIN {X 0,Y 136.659,Z 906.935,A -85,B 0,C 180,E1 4887.734,E2 4887.734} C_VEL
LIN {X 0,Y 148.89,Z 896.433,A -85,B 0,C 180,E1 4884.058,E2 4884.058} C_VEL
LIN {X 0,Y 160.85,Z 884.464,A -85,B 0,C 180,E1 4881.211,E2 4881.211} C_VEL
LIN {X 0,Y 171.889,Z 871.478,A -85,B 0,C 180,E1 4879.075,E2 4879.075} C_VEL
LIN {X 0,Y 181.834,Z 857.556,A -85,B 0,C 180,E1 4877.469,E2 4877.469} C_VEL
LIN {X 0,Y 190.571,Z 842.623,A -85,B 0,C 180,E1 4876.263,E2 4876.263} C_VEL
LIN {X 0,Y 198.013,Z 826.775,A -85,B 0,C 180,E1 4875.356,E2 4875.356} C_VEL
LIN {X 0,Y 204.085,Z 809.874,A -85,B 0,C 180,E1 4874.659,E2 4874.659} C_VEL
LIN {X 0,Y 208.414,Z 792.514,A -85,B 0,C 180,E1 4874.142,E2 4874.142} C_VEL
LIN {X 0,Y 211.457,Z 771.235,A -85,B 0,C 180,E1 4873.675,E2 4873.675} C_VEL
LIN {X 0,Y 216.67,Z 726.52,A -85,B 0,C 180,E1 4872.729,E2 4872.729} C_VEL
LIN {X 0,Y 215.576,Z 723.638,A -85,B 0,C 180,E1 4869.342,E2 4869.342} C_VEL
LIN {X 0,Y 214.932,Z 723.032,A -85,B 0,C 180,E1 4865.07,E2 4865.07} C_VEL
LIN {X 0,Y 215.306,Z 725.55,A -85,B 0,C 180,E1 4860.532,E2 4860.532} C_VEL
LIN {X 0,Y 215.919,Z 728.824,A -85,B 0,C 180,E1 4857.89,E2 4857.89} C_VEL
LIN {X 0,Y 209.42,Z 781.497,A -85,B 0,C 180,E1 4856.692,E2 4856.692} C_VEL
LIN {X 0,Y 205.748,Z 798.478,A -85,B 0,C 180,E1 4856.014,E2 4856.014} C_VEL
LIN {X 0,Y 200.433,Z 815.074,A -85,B 0,C 180,E1 4855.072,E2 4855.072} C_VEL
LIN {X 0,Y 194.03,Z 829.918,A -85,B 0,C 180,E1 4853.935,E2 4853.935} C_VEL
LIN {X 0,Y 186.059,Z 844.378,A -85,B 0,C 180,E1 4852.45,E2 4852.45} C_VEL
LIN {X 0,Y 176.736,Z 858.055,A -85,B 0,C 180,E1 4850.557,E2 4850.557} C_VEL
LIN {X 0,Y 166.905,Z 869.901,A -85,B 0,C 180,E1 4848.323,E2 4848.323} C_VEL
LIN {X 0,Y 155.956,Z 880.791,A -85,B 0,C 180,E1 4845.449,E2 4845.449} C_VEL
LIN {X 0,Y 144.56,Z 890.227,A -85,B 0,C 180,E1 4841.865,E2 4841.865} C_VEL
LIN {X 0,Y 133.27,Z 897.904,A -85,B 0,C 180,E1 4837.502,E2 4837.502} C_VEL
LIN {X 0,Y 122.224,Z 903.953,A -85,B 0,C 180,E1 4832.046,E2 4832.046} C_VEL
LIN {X 0,Y 111.956,Z 908.336,A -85,B 0,C 180,E1 4825.231,E2 4825.231} C_VEL
LIN {X 0,Y 103.484,Z 910.719,A -85,B 0,C 180,E1 4817.234,E2 4817.234} C_VEL
LIN {X 0,Y 96.899,Z 911.297,A -85,B 0,C 180,E1 4807.49,E2 4807.49} C_VEL
LIN {X 0,Y 93.275,Z 910.018,A -85,B 0,C 180,E1 4797.436,E2 4797.436} C_VEL
LIN {X 0,Y 92.23,Z 906.98,A -85,B 0,C 180,E1 4787.011,E2 4787.011} C_VEL
LIN {X 0,Y 93.69,Z 902.193,A -85,B 0,C 180,E1 4776.733,E2 4776.733} C_VEL
LIN {X 0,Y 97.208,Z 895.896,A -85,B 0,C 180,E1 4767.635,E2 4767.635} C_VEL
LIN {X 0,Y 102.852,Z 887.379,A -85,B 0,C 180,E1 4759.074,E2 4759.074} C_VEL
LIN {X 0,Y 109.252,Z 877.938,A -85,B 0,C 180,E1 4752.416,E2 4752.416} C_VEL
LIN {X 0,Y 116.471,Z 866.612,A -85,B 0,C 180,E1 4746.736,E2 4746.736} C_VEL
LIN {X 0,Y 123.581,Z 854.308,A -85,B 0,C 180,E1 4742.272,E2 4742.272} C_VEL
LIN {X 0,Y 130.133,Z 841.224,A -85,B 0,C 180,E1 4738.805,E2 4738.805} C_VEL
LIN {X 0,Y 136.393,Z 826.381,A -85,B 0,C 180,E1 4735.934,E2 4735.934} C_VEL
LIN {X 0,Y 141.456,Z 811.533,A -85,B 0,C 180,E1 4733.826,E2 4733.826} C_VEL
LIN {X 0,Y 145.682,Z 794.982,A -85,B 0,C 180,E1 4732.162,E2 4732.162} C_VEL
LIN {X 0,Y 148.698,Z 777.403,A -85,B 0,C 180,E1 4730.982,E2 4730.982} C_VEL
LIN {X 0,Y 154.938,Z 713.53,A -85,B 0,C 180,E1 4728.756,E2 4728.756} C_VEL
LIN {X 0,Y 156.561,Z 695.593,A -85,B 0,C 180,E1 4728.123,E2 4728.123} C_VEL
LIN {X 0,Y 156.21,Z 679.711,A -85,B 0,C 180,E1 4726.46,E2 4726.46} C_VEL
LIN {X 0,Y 151.934,Z 668.448,A -85,B 0,C 180,E1 4722.292,E2 4722.292} C_VEL
LIN {X 0,Y 148.185,Z 660.012,A -85,B 0,C 180,E1 4718.004,E2 4718.004} C_VEL
LIN {X 0,Y 144.52,Z 652.53,A -85,B 0,C 180,E1 4712.778,E2 4712.778} C_VEL
LIN {X 0,Y 141.724,Z 647.028,A -85,B 0,C 180,E1 4707.069,E2 4707.069} C_VEL
LIN {X 0,Y 140.36,Z 644.823,A -85,B 0,C 180,E1 4703.067,E2 4703.067} C_VEL
LIN {X 0,Y 139.536,Z 642.795,A -85,B 0,C 180,E1 4697.947,E2 4697.947} C_VEL
LIN {X 0,Y 139.818,Z 642.869,A -85,B 0,C 180,E1 4690.716,E2 4690.716} C_VEL
LIN {X 0,Y 140.86,Z 644.098,A -85,B 0,C 180,E1 4686.406,E2 4686.406} C_VEL
LIN {X 0,Y 143.099,Z 647.312,A -85,B 0,C 180,E1 4681.002,E2 4681.002} C_VEL
LIN {X 0,Y 146.293,Z 652.571,A -85,B 0,C 180,E1 4675.689,E2 4675.689} C_VEL
LIN {X 0,Y 149.828,Z 658.795,A -85,B 0,C 180,E1 4671.278,E2 4671.278} C_VEL
LIN {X 0,Y 153.807,Z 666.633,A -85,B 0,C 180,E1 4667.145,E2 4667.145} C_VEL
LIN {X 0,Y 157.92,Z 675.766,A -85,B 0,C 180,E1 4663.494,E2 4663.494} C_VEL
LIN {X 0,Y 160.656,Z 682.747,A -85,B 0,C 180,E1 4661.289,E2 4661.289} C_VEL
LIN {X 0,Y 150.396,Z 791.487,A -85,B 0,C 180,E1 4657.846,E2 4657.846} C_VEL
LIN {X 0,Y 147.127,Z 809.63,A -85,B 0,C 180,E1 4656.805,E2 4656.805} C_VEL
LIN {X 0,Y 142.453,Z 826.849,A -85,B 0,C 180,E1 4655.36,E2 4655.36} C_VEL
LIN {X 0,Y 136.468,Z 843.365,A -85,B 0,C 180,E1 4653.363,E2 4653.363} C_VEL
LIN {X 0,Y 129.57,Z 858.883,A -85,B 0,C 180,E1 4650.693,E2 4650.693} C_VEL
LIN {X 0,Y 121.98,Z 873.499,A -85,B 0,C 180,E1 4647.162,E2 4647.162} C_VEL
LIN {X 0,Y 114.132,Z 886.853,A -85,B 0,C 180,E1 4642.64,E2 4642.64} C_VEL
LIN {X 0,Y 106.587,Z 898.626,A -85,B 0,C 180,E1 4637.033,E2 4637.033} C_VEL
LIN {X 0,Y 99.278,Z 909.925,A -85,B 0,C 180,E1 4629.387,E2 4629.387} C_VEL
LIN {X 0,Y 93.945,Z 918.949,A -85,B 0,C 180,E1 4620.727,E2 4620.727} C_VEL
LIN {X 0,Y 90.783,Z 926.415,A -85,B 0,C 180,E1 4610.586,E2 4610.586} C_VEL
LIN {X 0,Y 90.414,Z 932.167,A -85,B 0,C 180,E1 4599.555,E2 4599.555} C_VEL
LIN {X 0,Y 92.288,Z 935.604,A -85,B 0,C 180,E1 4589.852,E2 4589.852} C_VEL
LIN {X 0,Y 90.074,Z 936.548,A -85,B 0,C 180,E1 4579.132,E2 4579.132} C_VEL
LIN {X 0,Y 90.606,Z 935.976,A -85,B 0,C 180,E1 4568.59,E2 4568.59} C_VEL
LIN {X 0,Y 90.866,Z 935.195,A -85,B 0,C 180,E1 4563.71,E2 4563.71} C_VEL
LIN {X 0,Y 91.093,Z 931.729,A -85,B 0,C 180,E1 4551.187,E2 4551.187} C_VEL
LIN {X 0,Y 93.629,Z 929.959,A -85,B 0,C 180,E1 4546.764,E2 4546.764} C_VEL
LIN {X 0,Y 103.941,Z 924.769,A -85,B 0,C 180,E1 4537.944,E2 4537.944} C_VEL
LIN {X 0,Y 115.867,Z 917.959,A -85,B 0,C 180,E1 4531.181,E2 4531.181} C_VEL
LIN {X 0,Y 128.16,Z 909.903,A -85,B 0,C 180,E1 4526.231,E2 4526.231} C_VEL
LIN {X 0,Y 140.618,Z 900.401,A -85,B 0,C 180,E1 4522.454,E2 4522.454} C_VEL
LIN {X 0,Y 152.768,Z 889.546,A -85,B 0,C 180,E1 4519.557,E2 4519.557} C_VEL
LIN {X 0,Y 164.868,Z 876.804,A -85,B 0,C 180,E1 4517.25,E2 4517.25} C_VEL
LIN {X 0,Y 175.875,Z 862.979,A -85,B 0,C 180,E1 4515.536,E2 4515.536} C_VEL
LIN {X 0,Y 185.197,Z 848.743,A -85,B 0,C 180,E1 4514.315,E2 4514.315} C_VEL
LIN {X 0,Y 193.683,Z 832.718,A -85,B 0,C 180,E1 4513.356,E2 4513.356} C_VEL
LIN {X 0,Y 200.321,Z 816.676,A -85,B 0,C 180,E1 4512.671,E2 4512.671} C_VEL
LIN {X 0,Y 205.476,Z 799.644,A -85,B 0,C 180,E1 4512.142,E2 4512.142} C_VEL
LIN {X 0,Y 208.959,Z 781.587,A -85,B 0,C 180,E1 4511.725,E2 4511.725} C_VEL
LIN {X 0,Y 214.9,Z 732.683,A -85,B 0,C 180,E1 4510.725,E2 4510.725} C_VEL
LIN {X 0,Y 214.307,Z 731.268,A -85,B 0,C 180,E1 4508.315,E2 4508.315} C_VEL
LIN {X 0,Y 213.889,Z 731.086,A -85,B 0,C 180,E1 4504.826,E2 4504.826} C_VEL
LIN {X 0,Y 214.18,Z 733.335,A -85,B 0,C 180,E1 4500.936,E2 4500.936} C_VEL
LIN {X 0,Y 214.317,Z 734.772,A -85,B 0,C 180,E1 4499.895,E2 4499.895} C_VEL
LIN {X 0,Y 208.263,Z 782.457,A -85,B 0,C 180,E1 4498.849,E2 4498.849} C_VEL
LIN {X 0,Y 204.448,Z 799.513,A -85,B 0,C 180,E1 4498.2,E2 4498.2} C_VEL
LIN {X 0,Y 198.913,Z 816.253,A -85,B 0,C 180,E1 4497.301,E2 4497.301} C_VEL
LIN {X 0,Y 192.003,Z 831.637,A -85,B 0,C 180,E1 4496.179,E2 4496.179} C_VEL
LIN {X 0,Y 183.713,Z 846.106,A -85,B 0,C 180,E1 4494.761,E2 4494.761} C_VEL
LIN {X 0,Y 174.249,Z 859.512,A -85,B 0,C 180,E1 4492.994,E2 4492.994} C_VEL
LIN {X 0,Y 164.033,Z 871.35,A -85,B 0,C 180,E1 4490.862,E2 4490.862} C_VEL
LIN {X 0,Y 153.167,Z 881.782,A -85,B 0,C 180,E1 4488.243,E2 4488.243} C_VEL
LIN {X 0,Y 141.307,Z 891.237,A -85,B 0,C 180,E1 4484.822,E2 4484.822} C_VEL
LIN {X 0,Y 129.42,Z 898.978,A -85,B 0,C 180,E1 4480.596,E2 4480.596} C_VEL
LIN {X 0,Y 117.754,Z 905.032,A -85,B 0,C 180,E1 4475.28,E2 4475.28} C_VEL
LIN {X 0,Y 106.703,Z 909.443,A -85,B 0,C 180,E1 4468.487,E2 4468.487} C_VEL
LIN {X 0,Y 97.4,Z 911.886,A -85,B 0,C 180,E1 4460.328,E2 4460.328} C_VEL
LIN {X 0,Y 89.969,Z 912.516,A -85,B 0,C 180,E1 4450.12,E2 4450.12} C_VEL
LIN {X 0,Y 85.71,Z 911.322,A -85,B 0,C 180,E1 4439.326,E2 4439.326} C_VEL
LIN {X 0,Y 84.282,Z 908.343,A -85,B 0,C 180,E1 4427.955,E2 4427.955} C_VEL
LIN {X 0,Y 85.65,Z 903.621,A -85,B 0,C 180,E1 4416.695,E2 4416.695} C_VEL
LIN {X 0,Y 89.321,Z 897.449,A -85,B 0,C 180,E1 4406.784,E2 4406.784} C_VEL
LIN {X 0,Y 95.159,Z 889.206,A -85,B 0,C 180,E1 4397.74,E2 4397.74} C_VEL
LIN {X 0,Y 102.063,Z 879.749,A -85,B 0,C 180,E1 4390.539,E2 4390.539} C_VEL
LIN {X 0,Y 109.68,Z 868.611,A -85,B 0,C 180,E1 4384.625,E2 4384.625} C_VEL
LIN {X 0,Y 117.485,Z 855.928,A -85,B 0,C 180,E1 4379.856,E2 4379.856} C_VEL
LIN {X 0,Y 124.429,Z 842.922,A -85,B 0,C 180,E1 4376.324,E2 4376.324} C_VEL
LIN {X 0,Y 130.974,Z 828.261,A -85,B 0,C 180,E1 4373.452,E2 4373.452} C_VEL
LIN {X 0,Y 136.564,Z 812.746,A -85,B 0,C 180,E1 4371.243,E2 4371.243} C_VEL
LIN {X 0,Y 141.001,Z 796.322,A -85,B 0,C 180,E1 4369.593,E2 4369.593} C_VEL
LIN {X 0,Y 144.242,Z 778.421,A -85,B 0,C 180,E1 4368.397,E2 4368.397} C_VEL
LIN {X 0,Y 149.947,Z 722.411,A -85,B 0,C 180,E1 4366.448,E2 4366.448} C_VEL
LIN {X 0,Y 152.443,Z 696.627,A -85,B 0,C 180,E1 4365.592,E2 4365.592} C_VEL
LIN {X 0,Y 152.285,Z 683.662,A -85,B 0,C 180,E1 4364.175,E2 4364.175} C_VEL
LIN {X 0,Y 148.874,Z 674.063,A -85,B 0,C 180,E1 4360.4,E2 4360.4} C_VEL
LIN {X 0,Y 145.384,Z 665.554,A -85,B 0,C 180,E1 4355.896,E2 4355.896} C_VEL
LIN {X 0,Y 142.545,Z 659.388,A -85,B 0,C 180,E1 4351.27,E2 4351.27} C_VEL
LIN {X 0,Y 140.187,Z 654.315,A -85,B 0,C 180,E1 4345.791,E2 4345.791} C_VEL
LIN {X 0,Y 138.548,Z 650.76,A -85,B 0,C 180,E1 4338.079,E2 4338.079} C_VEL
LIN {X 0,Y 138.802,Z 650.805,A -85,B 0,C 180,E1 4330.796,E2 4330.796} C_VEL
LIN {X 0,Y 139.719,Z 651.988,A -85,B 0,C 180,E1 4326.782,E2 4326.782} C_VEL
LIN {X 0,Y 141.642,Z 654.938,A -85,B 0,C 180,E1 4321.821,E2 4321.821} C_VEL
LIN {X 0,Y 144.515,Z 660.024,A -85,B 0,C 180,E1 4316.629,E2 4316.629} C_VEL
LIN {X 0,Y 147.632,Z 665.929,A -85,B 0,C 180,E1 4312.412,E2 4312.412} C_VEL
LIN {X 0,Y 151.409,Z 674,A -85,B 0,C 180,E1 4308.188,E2 4308.188} C_VEL
LIN {X 0,Y 155.403,Z 683.621,A -85,B 0,C 180,E1 4304.371,E2 4304.371} C_VEL
LIN {X 0,Y 156.16,Z 686.058,A -85,B 0,C 180,E1 4303.662,E2 4303.662} C_VEL
LIN {X 0,Y 145.866,Z 790.892,A -85,B 0,C 180,E1 4300.402,E2 4300.402} C_VEL
LIN {X 0,Y 142.455,Z 809.122,A -85,B 0,C 180,E1 4299.376,E2 4299.376} C_VEL
LIN {X 0,Y 137.757,Z 825.873,A -85,B 0,C 180,E1 4298.008,E2 4298.008} C_VEL
LIN {X 0,Y 131.756,Z 841.99,A -85,B 0,C 180,E1 4296.128,E2 4296.128} C_VEL
LIN {X 0,Y 124.562,Z 857.617,A -85,B 0,C 180,E1 4293.512,E2 4293.512} C_VEL
LIN {X 0,Y 116.596,Z 872.31,A -85,B 0,C 180,E1 4290.014,E2 4290.014} C_VEL
LIN {X 0,Y 108.641,Z 885.209,A -85,B 0,C 180,E1 4285.677,E2 4285.677} C_VEL
LIN {X 0,Y 100.533,Z 897.119,A -85,B 0,C 180,E1 4279.984,E2 4279.984} C_VEL
LIN {X 0,Y 93.037,Z 907.809,A -85,B 0,C 180,E1 4272.62,E2 4272.62} C_VEL
LIN {X 0,Y 86.96,Z 917.024,A -85,B 0,C 180,E1 4263.504,E2 4263.504} C_VEL
LIN {X 0,Y 83.148,Z 924.692,A -85,B 0,C 180,E1 4252.638,E2 4252.638} C_VEL
LIN {X 0,Y 82.337,Z 930.34,A -85,B 0,C 180,E1 4241.211,E2 4241.211} C_VEL
LIN {X 0,Y 84.219,Z 934.162,A -85,B 0,C 180,E1 4230.008,E2 4230.008} C_VEL
LIN {X 0,Y 82.274,Z 935.204,A -85,B 0,C 180,E1 4220.214,E2 4220.214} C_VEL
LIN {X 0,Y 82.865,Z 934.851,A -85,B 0,C 180,E1 4207.298,E2 4207.298} C_VEL
LIN {X 0,Y 87.828,Z 932.62,A -85,B 0,C 180,E1 4194.521,E2 4194.521} C_VEL
LIN {X 0,Y 93.629,Z 929.959,A -85,B 0,C 180,E1 4186.764,E2 4186.764} C_VEL
LIN {X 0,Y 96.689,Z 928.042,A -85,B 0,C 180,E1 4182.626,E2 4182.626} C_VEL
LIN {X 0,Y 103.598,Z 922.047,A -85,B 0,C 180,E1 4172.34,E2 4172.34} C_VEL
LIN {X 0,Y 108.117,Z 919.282,A -85,B 0,C 180,E1 4169.271,E2 4169.271} C_VEL
LIN {X 0,Y 121.421,Z 911.441,A -85,B 0,C 180,E1 4163.955,E2 4163.955} C_VEL
LIN {X 0,Y 135.085,Z 901.919,A -85,B 0,C 180,E1 4159.975,E2 4159.975} C_VEL
LIN {X 0,Y 148.439,Z 890.879,A -85,B 0,C 180,E1 4156.997,E2 4156.997} C_VEL
LIN {X 0,Y 160.805,Z 878.669,A -85,B 0,C 180,E1 4154.825,E2 4154.825} C_VEL
LIN {X 0,Y 172.01,Z 865.406,A -85,B 0,C 180,E1 4153.223,E2 4153.223} C_VEL
LIN {X 0,Y 182.429,Z 850.502,A -85,B 0,C 180,E1 4151.993,E2 4151.993} C_VEL
LIN {X 0,Y 191.038,Z 835.305,A -85,B 0,C 180,E1 4151.129,E2 4151.129} C_VEL
LIN {X 0,Y 198.247,Z 818.969,A -85,B 0,C 180,E1 4150.475,E2 4150.475} C_VEL
LIN {X 0,Y 203.987,Z 801.406,A -85,B 0,C 180,E1 4149.963,E2 4149.963} C_VEL
LIN {X 0,Y 207.757,Z 783.889,A -85,B 0,C 180,E1 4149.579,E2 4149.579} C_VEL
LIN {X 0,Y 213.38,Z 739.35,A -85,B 0,C 180,E1 4148.759,E2 4148.759} C_VEL
LIN {X 0,Y 212.882,Z 738.951,A -85,B 0,C 180,E1 4145.119,E2 4145.119} C_VEL
LIN {X 0,Y 212.983,Z 740.702,A -85,B 0,C 180,E1 4141.928,E2 4141.928} C_VEL
LIN {X 0,Y 207.411,Z 783.4,A -85,B 0,C 180,E1 4141.027,E2 4141.027} C_VEL
LIN {X 0,Y 203.478,Z 800.509,A -85,B 0,C 180,E1 4140.413,E2 4140.413} C_VEL
LIN {X 0,Y 197.947,Z 816.864,A -85,B 0,C 180,E1 4139.594,E2 4139.594} C_VEL
LIN {X 0,Y 191.004,Z 832.102,A -85,B 0,C 180,E1 4138.57,E2 4138.57} C_VEL
LIN {X 0,Y 182.527,Z 846.642,A -85,B 0,C 180,E1 4137.259,E2 4137.259} C_VEL
LIN {X 0,Y 173.217,Z 859.58,A -85,B 0,C 180,E1 4135.696,E2 4135.696} C_VEL
LIN {X 0,Y 162.914,Z 871.391,A -85,B 0,C 180,E1 4133.767,E2 4133.767} C_VEL
LIN {X 0,Y 151.286,Z 882.327,A -85,B 0,C 180,E1 4131.256,E2 4131.256} C_VEL
LIN {X 0,Y 138.452,Z 892.243,A -85,B 0,C 180,E1 4127.91,E2 4127.91} C_VEL
LIN {X 0,Y 125.928,Z 900.075,A -85,B 0,C 180,E1 4123.853,E2 4123.853} C_VEL
LIN {X 0,Y 113.69,Z 906.111,A -85,B 0,C 180,E1 4118.755,E2 4118.755} C_VEL
LIN {X 0,Y 101.83,Z 910.557,A -85,B 0,C 180,E1 4112.067,E2 4112.067} C_VEL
LIN {X 0,Y 91.64,Z 913.062,A -85,B 0,C 180,E1 4103.822,E2 4103.822} C_VEL
LIN {X 0,Y 83.259,Z 913.737,A -85,B 0,C 180,E1 4093.181,E2 4093.181} C_VEL
LIN {X 0,Y 78.249,Z 912.612,A -85,B 0,C 180,E1 4081.58,E2 4081.58} C_VEL
LIN {X 0,Y 76.359,Z 909.706,A -85,B 0,C 180,E1 4069.097,E2 4069.097} C_VEL
LIN {X 0,Y 77.609,Z 905.051,A -85,B 0,C 180,E1 4056.649,E2 4056.649} C_VEL
LIN {X 0,Y 81.455,Z 898.992,A -85,B 0,C 180,E1 4045.768,E2 4045.768} C_VEL
LIN {X 0,Y 87.569,Z 890.981,A -85,B 0,C 180,E1 4036.12,E2 4036.12} C_VEL
LIN {X 0,Y 94.998,Z 881.521,A -85,B 0,C 180,E1 4028.379,E2 4028.379} C_VEL
LIN {X 0,Y 103.058,Z 870.609,A -85,B 0,C 180,E1 4022.24,E2 4022.24} C_VEL
LIN {X 0,Y 111.265,Z 858.122,A -85,B 0,C 180,E1 4017.368,E2 4017.368} C_VEL
LIN {X 0,Y 118.909,Z 844.708,A -85,B 0,C 180,E1 4013.64,E2 4013.64} C_VEL
LIN {X 0,Y 125.75,Z 830.313,A -85,B 0,C 180,E1 4010.79,E2 4010.79} C_VEL
LIN {X 0,Y 131.971,Z 813.958,A -85,B 0,C 180,E1 4008.473,E2 4008.473} C_VEL
LIN {X 0,Y 136.622,Z 797.667,A -85,B 0,C 180,E1 4006.855,E2 4006.855} C_VEL
LIN {X 0,Y 140.027,Z 779.906,A -85,B 0,C 180,E1 4005.679,E2 4005.679} C_VEL
LIN {X 0,Y 144.18,Z 741.153,A -85,B 0,C 180,E1 4004.28,E2 4004.28} C_VEL
LIN {X 0,Y 148.639,Z 697.704,A -85,B 0,C 180,E1 4002.93,E2 4002.93} C_VEL
LIN {X 0,Y 148.608,Z 687.599,A -85,B 0,C 180,E1 4001.767,E2 4001.767} C_VEL
LIN {X 0,Y 145.684,Z 678.975,A -85,B 0,C 180,E1 3998.08,E2 3998.08} C_VEL
LIN {X 0,Y 142.824,Z 671.488,A -85,B 0,C 180,E1 3993.819,E2 3993.819} C_VEL
LIN {X 0,Y 140.721,Z 666.364,A -85,B 0,C 180,E1 3989.827,E2 3989.827} C_VEL
LIN {X 0,Y 138.784,Z 661.759,A -85,B 0,C 180,E1 3984.7,E2 3984.7} C_VEL
LIN {X 0,Y 137.493,Z 658.612,A -85,B 0,C 180,E1 3977.348,E2 3977.348} C_VEL
LIN {X 0,Y 137.856,Z 658.809,A -85,B 0,C 180,E1 3970.448,E2 3970.448} C_VEL
LIN {X 0,Y 138.618,Z 659.941,A -85,B 0,C 180,E1 3967.044,E2 3967.044} C_VEL
LIN {X 0,Y 140.201,Z 662.557,A -85,B 0,C 180,E1 3962.658,E2 3962.658} C_VEL
LIN {X 0,Y 142.721,Z 667.358,A -85,B 0,C 180,E1 3957.692,E2 3957.692} C_VEL
LIN {X 0,Y 145.484,Z 673.079,A -85,B 0,C 180,E1 3953.589,E2 3953.589} C_VEL
LIN {X 0,Y 149.139,Z 681.505,A -85,B 0,C 180,E1 3949.181,E2 3949.181} C_VEL
LIN {X 0,Y 151.974,Z 689.067,A -85,B 0,C 180,E1 3946.178,E2 3946.178} C_VEL
LIN {X 0,Y 141.652,Z 790.245,A -85,B 0,C 180,E1 3943.118,E2 3943.118} C_VEL
LIN {X 0,Y 138.119,Z 808.487,A -85,B 0,C 180,E1 3942.124,E2 3942.124} C_VEL
LIN {X 0,Y 133.137,Z 825.615,A -85,B 0,C 180,E1 3940.77,E2 3940.77} C_VEL
LIN {X 0,Y 126.95,Z 841.528,A -85,B 0,C 180,E1 3938.958,E2 3938.958} C_VEL
LIN {X 0,Y 119.473,Z 857.083,A -85,B 0,C 180,E1 3936.407,E2 3936.407} C_VEL
LIN {X 0,Y 111.143,Z 871.709,A -85,B 0,C 180,E1 3932.955,E2 3932.955} C_VEL
LIN {X 0,Y 102.598,Z 884.777,A -85,B 0,C 180,E1 3928.513,E2 3928.513} C_VEL
LIN {X 0,Y 93.968,Z 896.613,A -85,B 0,C 180,E1 3922.664,E2 3922.664} C_VEL
LIN {X 0,Y 85.569,Z 907.715,A -85,B 0,C 180,E1 3914.521,E2 3914.521} C_VEL
LIN {X 0,Y 79.11,Z 916.753,A -85,B 0,C 180,E1 3904.67,E2 3904.67} C_VEL
LIN {X 0,Y 75.129,Z 924.174,A -85,B 0,C 180,E1 3892.711,E2 3892.711} C_VEL
LIN {X 0,Y 74.465,Z 929.647,A -85,B 0,C 180,E1 3880.061,E2 3880.061} C_VEL
LIN {X 0,Y 76.239,Z 932.843,A -85,B 0,C 180,E1 3869.634,E2 3869.634} C_VEL
LIN {X 0,Y 74.139,Z 933.946,A -85,B 0,C 180,E1 3855.962,E2 3855.962} C_VEL
LIN {X 0,Y 76.47,Z 933.26,A -85,B 0,C 180,E1 3841.081,E2 3841.081} C_VEL
LIN {X 0,Y 83.551,Z 930.68,A -85,B 0,C 180,E1 3827.937,E2 3827.937} C_VEL
LIN {X 0,Y 93.751,Z 926.377,A -85,B 0,C 180,E1 3817.906,E2 3817.906} C_VEL
LIN {X 0,Y 106.341,Z 920.204,A -85,B 0,C 180,E1 3810.137,E2 3810.137} C_VEL
LIN {X 0,Y 108.117,Z 919.282,A -85,B 0,C 180,E1 3809.271,E2 3809.271} C_VEL
LIN {X 0,Y 112.902,Z 916.307,A -85,B 0,C 180,E1 3806.497,E2 3806.497} C_VEL
LIN {X 0,Y 123.659,Z 907.777,A -85,B 0,C 180,E1 3799.371,E2 3799.371} C_VEL
LIN {X 0,Y 128.977,Z 903.923,A -85,B 0,C 180,E1 3797.492,E2 3797.492} C_VEL
LIN {X 0,Y 142.574,Z 893.651,A -85,B 0,C 180,E1 3794.622,E2 3794.622} C_VEL
LIN {X 0,Y 155.631,Z 881.787,A -85,B 0,C 180,E1 3792.481,E2 3792.481} C_VEL
LIN {X 0,Y 167.962,Z 868.366,A -85,B 0,C 180,E1 3790.868,E2 3790.868} C_VEL
LIN {X 0,Y 178.522,Z 854.448,A -85,B 0,C 180,E1 3789.743,E2 3789.743} C_VEL
LIN {X 0,Y 187.716,Z 839.469,A -85,B 0,C 180,E1 3788.92,E2 3788.92} C_VEL
LIN {X 0,Y 195.495,Z 823.527,A -85,B 0,C 180,E1 3788.309,E2 3788.309} C_VEL
LIN {X 0,Y 201.581,Z 807.172,A -85,B 0,C 180,E1 3787.85,E2 3787.85} C_VEL
LIN {X 0,Y 206.054,Z 789.832,A -85,B 0,C 180,E1 3787.482,E2 3787.482} C_VEL
LIN {X 0,Y 209.534,Z 766.392,A -85,B 0,C 180,E1 3787.071,E2 3787.071} C_VEL
LIN {X 0,Y 211.994,Z 746.887,A -85,B 0,C 180,E1 3786.703,E2 3786.703} C_VEL
LIN {X 0,Y 211.829,Z 747.075,A -85,B 0,C 180,E1 3784.873,E2 3784.873} C_VEL
LIN {X 0,Y 211.776,Z 747.753,A -85,B 0,C 180,E1 3783.964,E2 3783.964} C_VEL
LIN {X 0,Y 206.826,Z 784.525,A -85,B 0,C 180,E1 3783.215,E2 3783.215} C_VEL
LIN {X 0,Y 202.743,Z 801.745,A -85,B 0,C 180,E1 3782.635,E2 3782.635} C_VEL
LIN {X 0,Y 197.048,Z 818.133,A -85,B 0,C 180,E1 3781.871,E2 3781.871} C_VEL
LIN {X 0,Y 189.766,Z 833.614,A -85,B 0,C 180,E1 3780.905,E2 3780.905} C_VEL
LIN {X 0,Y 180.949,Z 848.294,A -85,B 0,C 180,E1 3779.677,E2 3779.677} C_VEL
LIN {X 0,Y 171.036,Z 861.613,A -85,B 0,C 180,E1 3778.174,E2 3778.174} C_VEL
LIN {X 0,Y 159.79,Z 873.869,A -85,B 0,C 180,E1 3776.268,E2 3776.268} C_VEL
LIN {X 0,Y 147.791,Z 884.589,A -85,B 0,C 180,E1 3773.898,E2 3773.898} C_VEL
LIN {X 0,Y 135.622,Z 893.542,A -85,B 0,C 180,E1 3771.012,E2 3771.012} C_VEL
LIN {X 0,Y 122.962,Z 901.123,A -85,B 0,C 180,E1 3767.314,E2 3767.314} C_VEL
LIN {X 0,Y 110.075,Z 907.188,A -85,B 0,C 180,E1 3762.471,E2 3762.471} C_VEL
LIN {X 0,Y 97.396,Z 911.67,A -85,B 0,C 180,E1 3755.989,E2 3755.989} C_VEL
LIN {X 0,Y 86.267,Z 914.239,A -85,B 0,C 180,E1 3747.766,E2 3747.766} C_VEL
LIN {X 0,Y 76.828,Z 914.959,A -85,B 0,C 180,E1 3736.767,E2 3736.767} C_VEL
LIN {X 0,Y 70.932,Z 913.882,A -85,B 0,C 180,E1 3724.306,E2 3724.306} C_VEL
LIN {X 0,Y 68.468,Z 911.058,A -85,B 0,C 180,E1 3710.504,E2 3710.504} C_VEL
LIN {X 0,Y 69.562,Z 906.468,A -85,B 0,C 180,E1 3696.592,E2 3696.592} C_VEL
LIN {X 0,Y 73.981,Z 900.044,A -85,B 0,C 180,E1 3683.784,E2 3683.784} C_VEL
LIN {X 0,Y 80.675,Z 892.015,A -85,B 0,C 180,E1 3673.43,E2 3673.43} C_VEL
LIN {X 0,Y 88.712,Z 882.552,A -85,B 0,C 180,E1 3665.347,E2 3665.347} C_VEL
LIN {X 0,Y 97.333,Z 871.643,A -85,B 0,C 180,E1 3659.089,E2 3659.089} C_VEL
LIN {X 0,Y 106.028,Z 859.165,A -85,B 0,C 180,E1 3654.216,E2 3654.216} C_VEL
LIN {X 0,Y 114.027,Z 845.844,A -85,B 0,C 180,E1 3650.555,E2 3650.555} C_VEL
LIN {X 0,Y 121.222,Z 831.447,A -85,B 0,C 180,E1 3647.758,E2 3647.758} C_VEL
LIN {X 0,Y 127.707,Z 815.17,A -85,B 0,C 180,E1 3645.512,E2 3645.512} C_VEL
LIN {X 0,Y 132.64,Z 798.739,A -85,B 0,C 180,E1 3643.922,E2 3643.922} C_VEL
LIN {X 0,Y 136.196,Z 781.079,A -85,B 0,C 180,E1 3642.783,E2 3642.783} C_VEL
LIN {X 0,Y 139.78,Z 749.265,A -85,B 0,C 180,E1 3641.624,E2 3641.624} C_VEL
LIN {X 0,Y 145.175,Z 698.595,A -85,B 0,C 180,E1 3640.115,E2 3640.115} C_VEL
LIN {X 0,Y 145.221,Z 691.798,A -85,B 0,C 180,E1 3639.305,E2 3639.305} C_VEL
LIN {X 0,Y 142.931,Z 684.481,A -85,B 0,C 180,E1 3635.989,E2 3635.989} C_VEL
LIN {X 0,Y 140.625,Z 677.823,A -85,B 0,C 180,E1 3631.986,E2 3631.986} C_VEL
LIN {X 0,Y 139.071,Z 673.588,A -85,B 0,C 180,E1 3628.563,E2 3628.563} C_VEL
LIN {X 0,Y 137.419,Z 669.168,A -85,B 0,C 180,E1 3623.54,E2 3623.54} C_VEL
LIN {X 0,Y 136.475,Z 666.523,A -85,B 0,C 180,E1 3617.042,E2 3617.042} C_VEL
LIN {X 0,Y 136.916,Z 666.83,A -85,B 0,C 180,E1 3610.095,E2 3610.095} C_VEL
LIN {X 0,Y 137.886,Z 668.562,A -85,B 0,C 180,E1 3606.036,E2 3606.036} C_VEL
LIN {X 0,Y 138.862,Z 670.367,A -85,B 0,C 180,E1 3603.303,E2 3603.303} C_VEL
LIN {X 0,Y 141.016,Z 674.772,A -85,B 0,C 180,E1 3598.71,E2 3598.71} C_VEL
LIN {X 0,Y 143.535,Z 680.537,A -85,B 0,C 180,E1 3594.604,E2 3594.604} C_VEL
LIN {X 0,Y 146.789,Z 688.727,A -85,B 0,C 180,E1 3590.345,E2 3590.345} C_VEL
LIN {X 0,Y 148.03,Z 692.719,A -85,B 0,C 180,E1 3588.815,E2 3588.815} C_VEL
LIN {X 0,Y 137.762,Z 789.678,A -85,B 0,C 180,E1 3585.99,E2 3585.99} C_VEL
LIN {X 0,Y 134.12,Z 807.846,A -85,B 0,C 180,E1 3585.044,E2 3585.044} C_VEL
LIN {X 0,Y 129.116,Z 824.555,A -85,B 0,C 180,E1 3583.792,E2 3583.792} C_VEL
LIN {X 0,Y 122.915,Z 840.122,A -85,B 0,C 180,E1 3582.13,E2 3582.13} C_VEL
LIN {X 0,Y 115.141,Z 855.774,A -85,B 0,C 180,E1 3579.698,E2 3579.698} C_VEL
LIN {X 0,Y 106.418,Z 870.466,A -85,B 0,C 180,E1 3576.363,E2 3576.363} C_VEL
LIN {X 0,Y 97.392,Z 883.593,A -85,B 0,C 180,E1 3572,E2 3572} C_VEL
LIN {X 0,Y 88.019,Z 895.638,A -85,B 0,C 180,E1 3566.029,E2 3566.029} C_VEL
LIN {X 0,Y 79.32,Z 906.233,A -85,B 0,C 180,E1 3558.057,E2 3558.057} C_VEL
LIN {X 0,Y 72.075,Z 915.344,A -85,B 0,C 180,E1 3547.626,E2 3547.626} C_VEL
LIN {X 0,Y 67.436,Z 922.847,A -85,B 0,C 180,E1 3534.538,E2 3534.538} C_VEL
LIN {X 0,Y 66.491,Z 928.372,A -85,B 0,C 180,E1 3520.406,E2 3520.406} C_VEL
LIN {X 0,Y 68.099,Z 931.489,A -85,B 0,C 180,E1 3509.169,E2 3509.169} C_VEL
LIN {X 0,Y 66.286,Z 932.643,A -85,B 0,C 180,E1 3493.358,E2 3493.358} C_VEL
LIN {X 0,Y 69.718,Z 931.974,A -85,B 0,C 180,E1 3476.992,E2 3476.992} C_VEL
LIN {X 0,Y 78.195,Z 929.423,A -85,B 0,C 180,E1 3463.229,E2 3463.229} C_VEL
LIN {X 0,Y 90.09,Z 924.956,A -85,B 0,C 180,E1 3452.943,E2 3452.943} C_VEL
LIN {X 0,Y 104.076,Z 918.613,A -85,B 0,C 180,E1 3445.463,E2 3445.463} C_VEL
LIN {X 0,Y 118.343,Z 910.802,A -85,B 0,C 180,E1 3440.342,E2 3440.342} C_VEL
LIN {X 0,Y 128.977,Z 903.923,A -85,B 0,C 180,E1 3437.492,E2 3437.492} C_VEL
LIN {X 0,Y 134.357,Z 899.896,A -85,B 0,C 180,E1 3435.795,E2 3435.795} C_VEL
LIN {X 0,Y 146.351,Z 888.827,A -85,B 0,C 180,E1 3430.998,E2 3430.998} C_VEL
LIN {X 0,Y 151.604,Z 883.934,A -85,B 0,C 180,E1 3429.867,E2 3429.867} C_VEL
LIN {X 0,Y 164.21,Z 871.145,A -85,B 0,C 180,E1 3428.402,E2 3428.402} C_VEL
LIN {X 0,Y 175.391,Z 857.313,A -85,B 0,C 180,E1 3427.354,E2 3427.354} C_VEL
LIN {X 0,Y 185.173,Z 842.499,A -85,B 0,C 180,E1 3426.601,E2 3426.601} C_VEL
LIN {X 0,Y 193.521,Z 826.639,A -85,B 0,C 180,E1 3426.05,E2 3426.05} C_VEL
LIN {X 0,Y 200.159,Z 810.005,A -85,B 0,C 180,E1 3425.634,E2 3425.634} C_VEL
LIN {X 0,Y 205.192,Z 792.349,A -85,B 0,C 180,E1 3425.297,E2 3425.297} C_VEL
LIN {X 0,Y 205.478,Z 791.143,A -85,B 0,C 180,E1 3425.26,E2 3425.26} C_VEL
LIN {X 0,Y 200.865,Z 807.635,A -85,B 0,C 180,E1 3424.691,E2 3424.691} C_VEL
LIN {X 0,Y 194.4,Z 824.038,A -85,B 0,C 180,E1 3423.926,E2 3423.926} C_VEL
LIN {X 0,Y 186.753,Z 838.892,A -85,B 0,C 180,E1 3423.011,E2 3423.011} C_VEL
LIN {X 0,Y 177.54,Z 853.002,A -85,B 0,C 180,E1 3421.853,E2 3421.853} C_VEL
LIN {X 0,Y 166.577,Z 866.522,A -85,B 0,C 180,E1 3420.343,E2 3420.343} C_VEL
LIN {X 0,Y 154.925,Z 878.264,A -85,B 0,C 180,E1 3418.52,E2 3418.52} C_VEL
LIN {X 0,Y 142.269,Z 888.625,A -85,B 0,C 180,E1 3416.195,E2 3416.195} C_VEL
LIN {X 0,Y 128.868,Z 897.519,A -85,B 0,C 180,E1 3413.19,E2 3413.19} C_VEL
LIN {X 0,Y 114.981,Z 904.879,A -85,B 0,C 180,E1 3409.246,E2 3409.246} C_VEL
LIN {X 0,Y 101.765,Z 910.209,A -85,B 0,C 180,E1 3404.295,E2 3404.295} C_VEL
LIN {X 0,Y 88.662,Z 913.985,A -85,B 0,C 180,E1 3397.453,E2 3397.453} C_VEL
LIN {X 0,Y 77.302,Z 915.915,A -85,B 0,C 180,E1 3388.588,E2 3388.588} C_VEL
LIN {X 0,Y 68.225,Z 916.054,A -85,B 0,C 180,E1 3377.099,E2 3377.099} C_VEL
LIN {X 0,Y 62.142,Z 914.311,A -85,B 0,C 180,E1 3362.054,E2 3362.054} C_VEL
LIN {X 0,Y 60.483,Z 910.936,A -85,B 0,C 180,E1 3346.308,E2 3346.308} C_VEL
LIN {X 0,Y 62.859,Z 905.719,A -85,B 0,C 180,E1 3330.9,E2 3330.9} C_VEL
LIN {X 0,Y 68.806,Z 898.604,A -85,B 0,C 180,E1 3317.401,E2 3317.401} C_VEL
LIN {X 0,Y 76.326,Z 890.551,A -85,B 0,C 180,E1 3307.665,E2 3307.665} C_VEL
LIN {X 0,Y 85.445,Z 880.396,A -85,B 0,C 180,E1 3299.783,E2 3299.783} C_VEL
LIN {X 0,Y 94.937,Z 868.752,A -85,B 0,C 180,E1 3293.853,E2 3293.853} C_VEL
LIN {X 0,Y 103.821,Z 856.143,A -85,B 0,C 180,E1 3289.538,E2 3289.538} C_VEL
LIN {X 0,Y 112.465,Z 841.559,A -85,B 0,C 180,E1 3286.092,E2 3286.092} C_VEL
LIN {X 0,Y 119.582,Z 826.931,A -85,B 0,C 180,E1 3283.673,E2 3283.673} C_VEL
LIN {X 0,Y 125.497,Z 811.389,A -85,B 0,C 180,E1 3281.844,E2 3281.844} C_VEL
LIN {X 0,Y 130.358,Z 794.148,A -85,B 0,C 180,E1 3280.423,E2 3280.423} C_VEL
LIN {X 0,Y 133.466,Z 777.017,A -85,B 0,C 180,E1 3279.498,E2 3279.498} C_VEL
LIN {X 0,Y 142.007,Z 699.632,A -85,B 0,C 180,E1 3277.196,E2 3277.196} C_VEL
LIN {X 0,Y 142.046,Z 695.851,A -85,B 0,C 180,E1 3276.694,E2 3276.694} C_VEL
LIN {X 0,Y 139.889,Z 688.424,A -85,B 0,C 180,E1 3272.904,E2 3272.904} C_VEL
LIN {X 0,Y 138.345,Z 683.471,A -85,B 0,C 180,E1 3269.556,E2 3269.556} C_VEL
LIN {X 0,Y 137.204,Z 680.113,A -85,B 0,C 180,E1 3266.511,E2 3266.511} C_VEL
LIN {X 0,Y 136.172,Z 676.833,A -85,B 0,C 180,E1 3262.675,E2 3262.675} C_VEL
LIN {X 0,Y 135.462,Z 674.435,A -85,B 0,C 180,E1 3256.731,E2 3256.731} C_VEL
LIN {X 0,Y 135.898,Z 674.775,A -85,B 0,C 180,E1 3250.171,E2 3250.171} C_VEL
LIN {X 0,Y 137.328,Z 677.595,A -85,B 0,C 180,E1 3244.595,E2 3244.595} C_VEL
LIN {X 0,Y 139.281,Z 682.033,A -85,B 0,C 180,E1 3239.898,E2 3239.898} C_VEL
LIN {X 0,Y 141.569,Z 687.823,A -85,B 0,C 180,E1 3235.748,E2 3235.748} C_VEL
LIN {X 0,Y 144.349,Z 695.747,A -85,B 0,C 180,E1 3231.687,E2 3231.687} C_VEL
LIN {X 0,Y 134.25,Z 788.918,A -85,B 0,C 180,E1 3229.024,E2 3229.024} C_VEL
LIN {X 0,Y 130.518,Z 807.041,A -85,B 0,C 180,E1 3228.142,E2 3228.142} C_VEL
LIN {X 0,Y 125.224,Z 824.211,A -85,B 0,C 180,E1 3226.94,E2 3226.94} C_VEL
LIN {X 0,Y 118.422,Z 840.507,A -85,B 0,C 180,E1 3225.282,E2 3225.282} C_VEL
LIN {X 0,Y 110.334,Z 856.009,A -85,B 0,C 180,E1 3222.957,E2 3222.957} C_VEL
LIN {X 0,Y 101.254,Z 870.508,A -85,B 0,C 180,E1 3219.741,E2 3219.741} C_VEL
LIN {X 0,Y 92.174,Z 882.926,A -85,B 0,C 180,E1 3215.658,E2 3215.658} C_VEL
LIN {X 0,Y 82.212,Z 894.896,A -85,B 0,C 180,E1 3209.72,E2 3209.72} C_VEL
LIN {X 0,Y 72.804,Z 905.434,A -85,B 0,C 180,E1 3201.528,E2 3201.528} C_VEL
LIN {X 0,Y 64.822,Z 914.49,A -85,B 0,C 180,E1 3190.389,E2 3190.389} C_VEL
LIN {X 0,Y 59.619,Z 921.91,A -85,B 0,C 180,E1 3175.862,E2 3175.862} C_VEL
LIN {X 0,Y 58.651,Z 927.658,A -85,B 0,C 180,E1 3158.837,E2 3158.837} C_VEL
LIN {X 0,Y 60.049,Z 930.065,A -85,B 0,C 180,E1 3149.058,E2 3149.058} C_VEL
LIN {X 0,Y 58.515,Z 931.329,A -85,B 0,C 180,E1 3131.07,E2 3131.07} C_VEL
LIN {X 0,Y 62.996,Z 930.766,A -85,B 0,C 180,E1 3112.923,E2 3112.923} C_VEL
LIN {X 0,Y 72.813,Z 928.338,A -85,B 0,C 180,E1 3098.512,E2 3098.512} C_VEL
LIN {X 0,Y 85.415,Z 924.223,A -85,B 0,C 180,E1 3088.631,E2 3088.631} C_VEL
LIN {X 0,Y 99.975,Z 918.196,A -85,B 0,C 180,E1 3081.582,E2 3081.582} C_VEL
LIN {X 0,Y 114.859,Z 910.623,A -85,B 0,C 180,E1 3076.79,E2 3076.79} C_VEL
LIN {X 0,Y 129.498,Z 901.54,A -85,B 0,C 180,E1 3073.426,E2 3073.426} C_VEL
LIN {X 0,Y 143.587,Z 890.917,A -85,B 0,C 180,E1 3070.987,E2 3070.987} C_VEL
LIN {X 0,Y 151.604,Z 883.934,A -85,B 0,C 180,E1 3069.867,E2 3069.867} C_VEL
LIN {X 0,Y 156.799,Z 878.855,A -85,B 0,C 180,E1 3068.844,E2 3068.844} C_VEL
LIN {X 0,Y 168.374,Z 865.353,A -85,B 0,C 180,E1 3065.54,E2 3065.54} C_VEL
LIN {X 0,Y 173.018,Z 859.495,A -85,B 0,C 180,E1 3064.852,E2 3064.852} C_VEL
LIN {X 0,Y 177.887,Z 852.924,A -85,B 0,C 180,E1 3064.513,E2 3064.513} C_VEL
LIN {X 0,Y 167.219,Z 866.046,A -85,B 0,C 180,E1 3063.254,E2 3063.254} C_VEL
LIN {X 0,Y 155.014,Z 878.307,A -85,B 0,C 180,E1 3061.623,E2 3061.623} C_VEL
LIN {X 0,Y 142.126,Z 888.862,A -85,B 0,C 180,E1 3059.596,E2 3059.596} C_VEL
LIN {X 0,Y 128.143,Z 898.02,A -85,B 0,C 180,E1 3056.923,E2 3056.923} C_VEL
LIN {X 0,Y 113.71,Z 905.516,A -85,B 0,C 180,E1 3053.422,E2 3053.422} C_VEL
LIN {X 0,Y 99.811,Z 911.045,A -85,B 0,C 180,E1 3048.963,E2 3048.963} C_VEL
LIN {X 0,Y 85.844,Z 914.935,A -85,B 0,C 180,E1 3042.719,E2 3042.719} C_VEL
LIN {X 0,Y 72.895,Z 917.05,A -85,B 0,C 180,E1 3033.963,E2 3033.963} C_VEL
LIN {X 0,Y 62.211,Z 917.301,A -85,B 0,C 180,E1 3021.931,E2 3021.931} C_VEL
LIN {X 0,Y 54.885,Z 915.606,A -85,B 0,C 180,E1 3005.639,E2 3005.639} C_VEL
LIN {X 0,Y 52.521,Z 912.286,A -85,B 0,C 180,E1 2987.718,E2 2987.718} C_VEL
LIN {X 0,Y 54.876,Z 907.162,A -85,B 0,C 180,E1 2969.987,E2 2969.987} C_VEL
LIN {X 0,Y 61.328,Z 900.121,A -85,B 0,C 180,E1 2954.869,E2 2954.869} C_VEL
LIN {X 0,Y 69.481,Z 892.185,A -85,B 0,C 180,E1 2944.415,E2 2944.415} C_VEL
LIN {X 0,Y 79.255,Z 882.18,A -85,B 0,C 180,E1 2936.276,E2 2936.276} C_VEL
LIN {X 0,Y 89.308,Z 870.683,A -85,B 0,C 180,E1 2930.34,E2 2930.34} C_VEL
LIN {X 0,Y 98.742,Z 858.206,A -85,B 0,C 180,E1 2926.077,E2 2926.077} C_VEL
LIN {X 0,Y 107.654,Z 844.046,A -85,B 0,C 180,E1 2922.796,E2 2922.796} C_VEL
LIN {X 0,Y 115.479,Z 828.88,A -85,B 0,C 180,E1 2920.361,E2 2920.361} C_VEL
LIN {X 0,Y 121.904,Z 812.918,A -85,B 0,C 180,E1 2918.563,E2 2918.563} C_VEL
LIN {X 0,Y 127.088,Z 795.352,A -85,B 0,C 180,E1 2917.193,E2 2917.193} C_VEL
LIN {X 0,Y 130.37,Z 778.287,A -85,B 0,C 180,E1 2916.313,E2 2916.313} C_VEL
LIN {X 0,Y 139.223,Z 700.558,A -85,B 0,C 180,E1 2914.139,E2 2914.139} C_VEL
LIN {X 0,Y 137.593,Z 693.946,A -85,B 0,C 180,E1 2910.577,E2 2910.577} C_VEL
LIN {X 0,Y 136.01,Z 688.225,A -85,B 0,C 180,E1 2906.174,E2 2906.174} C_VEL
LIN {X 0,Y 134.992,Z 684.575,A -85,B 0,C 180,E1 2901.966,E2 2901.966} C_VEL
LIN {X 0,Y 134.454,Z 682.348,A -85,B 0,C 180,E1 2896.401,E2 2896.401} C_VEL
LIN {X 0,Y 134.956,Z 682.822,A -85,B 0,C 180,E1 2889.812,E2 2889.812} C_VEL
LIN {X 0,Y 136.044,Z 685.401,A -85,B 0,C 180,E1 2885.272,E2 2885.272} C_VEL
LIN {X 0,Y 137.595,Z 689.264,A -85,B 0,C 180,E1 2881.146,E2 2881.146} C_VEL
LIN {X 0,Y 139.543,Z 694.807,A -85,B 0,C 180,E1 2877.126,E2 2877.126} C_VEL
LIN {X 0,Y 141.047,Z 699.976,A -85,B 0,C 180,E1 2874.483,E2 2874.483} C_VEL
LIN {X 0,Y 131.026,Z 788.491,A -85,B 0,C 180,E1 2872.191,E2 2872.191} C_VEL
LIN {X 0,Y 127.142,Z 806.701,A -85,B 0,C 180,E1 2871.369,E2 2871.369} C_VEL
LIN {X 0,Y 121.733,Z 823.679,A -85,B 0,C 180,E1 2870.277,E2 2870.277} C_VEL
LIN {X 0,Y 114.688,Z 840.001,A -85,B 0,C 180,E1 2868.757,E2 2868.757} C_VEL
LIN {X 0,Y 105.916,Z 856.151,A -85,B 0,C 180,E1 2866.499,E2 2866.499} C_VEL
LIN {X 0,Y 96.48,Z 870.46,A -85,B 0,C 180,E1 2863.466,E2 2863.466} C_VEL
LIN {X 0,Y 86.134,Z 883.676,A -85,B 0,C 180,E1 2859.15,E2 2859.15} C_VEL
LIN {X 0,Y 75.253,Z 895.794,A -85,B 0,C 180,E1 2852.909,E2 2852.909} C_VEL
LIN {X 0,Y 65.283,Z 905.987,A -85,B 0,C 180,E1 2844.277,E2 2844.277} C_VEL
LIN {X 0,Y 56.793,Z 914.629,A -85,B 0,C 180,E1 2832.002,E2 2832.002} C_VEL
LIN {X 0,Y 51.423,Z 921.751,A -85,B 0,C 180,E1 2815.338,E2 2815.338} C_VEL
LIN {X 0,Y 50.867,Z 926.941,A -85,B 0,C 180,E1 2796.786,E2 2796.786} C_VEL
LIN {X 0,Y 51.994,Z 928.59,A -85,B 0,C 180,E1 2788.912,E2 2788.912} C_VEL
LIN {X 0,Y 50.863,Z 930.012,A -85,B 0,C 180,E1 2768.085,E2 2768.085} C_VEL
LIN {X 0,Y 56.665,Z 929.56,A -85,B 0,C 180,E1 2747.914,E2 2747.914} C_VEL
LIN {X 0,Y 68.369,Z 927.162,A -85,B 0,C 180,E1 2732.757,E2 2732.757} C_VEL
LIN {X 0,Y 82.622,Z 923.005,A -85,B 0,C 180,E1 2723.148,E2 2723.148} C_VEL
LIN {X 0,Y 98.154,Z 916.995,A -85,B 0,C 180,E1 2716.796,E2 2716.796} C_VEL
LIN {X 0,Y 113.704,Z 909.453,A -85,B 0,C 180,E1 2712.608,E2 2712.608} C_VEL
LIN {X 0,Y 128.809,Z 900.411,A -85,B 0,C 180,E1 2709.722,E2 2709.722} C_VEL
LIN {X 0,Y 143.235,Z 889.792,A -85,B 0,C 180,E1 2707.665,E2 2707.665} C_VEL
LIN {X 0,Y 156.864,Z 877.639,A -85,B 0,C 180,E1 2706.181,E2 2706.181} C_VEL
LIN {X 0,Y 168.636,Z 864.937,A -85,B 0,C 180,E1 2705.172,E2 2705.172} C_VEL
LIN {X 0,Y 173.018,Z 859.495,A -85,B 0,C 180,E1 2704.852,E2 2704.852} C_VEL
LIN {X 0,Y 171.714,Z 861.01,A -85,B 0,C 180,E1 2704.527,E2 2704.527} C_VEL
LIN {X 0,Y 164.455,Z 869.333,A -85,B 0,C 180,E1 2704.131,E2 2704.131} C_VEL
LIN {X 0,Y 152.388,Z 881.164,A -85,B 0,C 180,E1 2704.064,E2 2704.064} C_VEL
LIN {X 0,Y 142.782,Z 889.188,A -85,B 0,C 180,E1 2704.442,E2 2704.442} C_VEL
LIN {X 0,Y 139.491,Z 891.675,A -85,B 0,C 180,E1 2704.73,E2 2704.73} C_VEL
LIN {X 0,Y 124.768,Z 901.706,A -85,B 0,C 180,E1 2706.525,E2 2706.525} C_VEL
LIN {X 0,Y 109.334,Z 910.267,A -85,B 0,C 180,E1 2709.084,E2 2709.084} C_VEL
LIN {X 0,Y 93.322,Z 917.332,A -85,B 0,C 180,E1 2712.899,E2 2712.899} C_VEL
LIN {X 0,Y 77.085,Z 922.826,A -85,B 0,C 180,E1 2718.92,E2 2718.92} C_VEL
LIN {X 0,Y 62.35,Z 926.487,A -85,B 0,C 180,E1 2728.15,E2 2728.15} C_VEL
LIN {X 0,Y 50.311,Z 928.433,A -85,B 0,C 180,E1 2742.692,E2 2742.692} C_VEL
LIN {X 0,Y 43.224,Z 928.593,A -85,B 0,C 180,E1 2765.414,E2 2765.414} C_VEL
LIN {X 0,Y 43.944,Z 927.065,A -85,B 0,C 180,E1 2789.038,E2 2789.038} C_VEL
LIN {X 0,Y 42.846,Z 922.476,A -85,B 0,C 180,E1 2811.028,E2 2811.028} C_VEL
LIN {X 0,Y 47.391,Z 916.182,A -85,B 0,C 180,E1 2830.862,E2 2830.862} C_VEL
LIN {X 0,Y 55.906,Z 908.232,A -85,B 0,C 180,E1 2845.37,E2 2845.37} C_VEL
LIN {X 0,Y 66.174,Z 898.841,A -85,B 0,C 180,E1 2855.049,E2 2855.049} C_VEL
LIN {X 0,Y 77.828,Z 887.236,A -85,B 0,C 180,E1 2861.943,E2 2861.943} C_VEL
LIN {X 0,Y 88.501,Z 875.034,A -85,B 0,C 180,E1 2866.326,E2 2866.326} C_VEL
LIN {X 0,Y 98.756,Z 861.106,A -85,B 0,C 180,E1 2869.501,E2 2869.501} C_VEL
LIN {X 0,Y 108.102,Z 845.788,A -85,B 0,C 180,E1 2871.766,E2 2871.766} C_VEL
LIN {X 0,Y 115.78,Z 830.205,A -85,B 0,C 180,E1 2873.285,E2 2873.285} C_VEL
LIN {X 0,Y 122.07,Z 813.467,A -85,B 0,C 180,E1 2874.384,E2 2874.384} C_VEL
LIN {X 0,Y 126.827,Z 795.489,A -85,B 0,C 180,E1 2875.24,E2 2875.24} C_VEL
LIN {X 0,Y 129.69,Z 777.525,A -85,B 0,C 180,E1 2875.802,E2 2875.802} C_VEL
LIN {X 0,Y 138.048,Z 703.44,A -85,B 0,C 180,E1 2877.614,E2 2877.614} C_VEL
LIN {X 0,Y 136.328,Z 697.664,A -85,B 0,C 180,E1 2881.472,E2 2881.472} C_VEL
LIN {X 0,Y 135.232,Z 694.478,A -85,B 0,C 180,E1 2884.453,E2 2884.453} C_VEL
LIN {X 0,Y 134.28,Z 691.839,A -85,B 0,C 180,E1 2887.975,E2 2887.975} C_VEL
LIN {X 0,Y 133.684,Z 690.443,A -85,B 0,C 180,E1 2891.539,E2 2891.539} C_VEL
LIN {X 0,Y 133.458,Z 690.473,A -85,B 0,C 180,E1 2896.99,E2 2896.99} C_VEL
LIN {X 0,Y 134.003,Z 693.082,A -85,B 0,C 180,E1 2902.297,E2 2902.297} C_VEL
LIN {X 0,Y 134.992,Z 697.323,A -85,B 0,C 180,E1 2906.505,E2 2906.505} C_VEL
LIN {X 0,Y 136.195,Z 702.599,A -85,B 0,C 180,E1 2910.131,E2 2910.131} C_VEL
LIN {X 0,Y 136.54,Z 704.717,A -85,B 0,C 180,E1 2911.143,E2 2911.143} C_VEL
LIN {X 0,Y 127.639,Z 779.94,A -85,B 0,C 180,E1 2912.998,E2 2912.998} C_VEL
LIN {X 0,Y 124.017,Z 797.418,A -85,B 0,C 180,E1 2913.856,E2 2913.856} C_VEL
LIN {X 0,Y 118.862,Z 814.084,A -85,B 0,C 180,E1 2915.065,E2 2915.065} C_VEL
LIN {X 0,Y 112.243,Z 829.882,A -85,B 0,C 180,E1 2916.702,E2 2916.702} C_VEL
LIN {X 0,Y 104.126,Z 845.022,A -85,B 0,C 180,E1 2918.936,E2 2918.936} C_VEL
LIN {X 0,Y 94.827,Z 859.17,A -85,B 0,C 180,E1 2921.977,E2 2921.977} C_VEL
LIN {X 0,Y 84.655,Z 871.932,A -85,B 0,C 180,E1 2926.096,E2 2926.096} C_VEL
LIN {X 0,Y 74.203,Z 883.156,A -85,B 0,C 180,E1 2931.688,E2 2931.688} C_VEL
LIN {X 0,Y 63.614,Z 893.184,A -85,B 0,C 180,E1 2939.794,E2 2939.794} C_VEL
LIN {X 0,Y 54.002,Z 901.639,A -85,B 0,C 180,E1 2951.642,E2 2951.642} C_VEL
LIN {X 0,Y 46.908,Z 908.606,A -85,B 0,C 180,E1 2968.764,E2 2968.764} C_VEL
LIN {X 0,Y 44.599,Z 913.638,A -85,B 0,C 180,E1 2989.67,E2 2989.67} C_VEL
LIN {X 0,Y 48.29,Z 917.049,A -85,B 0,C 180,E1 3011.472,E2 3011.472} C_VEL
LIN {X 0,Y 56.732,Z 918.545,A -85,B 0,C 180,E1 3027.744,E2 3027.744} C_VEL
LIN {X 0,Y 68.624,Z 918.25,A -85,B 0,C 180,E1 3039.53,E2 3039.53} C_VEL
LIN {X 0,Y 82.826,Z 916.085,A -85,B 0,C 180,E1 3047.845,E2 3047.845} C_VEL
LIN {X 0,Y 97.76,Z 912.103,A -85,B 0,C 180,E1 3053.539,E2 3053.539} C_VEL
LIN {X 0,Y 112.101,Z 906.586,A -85,B 0,C 180,E1 3057.443,E2 3057.443} C_VEL
LIN {X 0,Y 126.964,Z 899.088,A -85,B 0,C 180,E1 3060.499,E2 3060.499} C_VEL
LIN {X 0,Y 141.41,Z 889.85,A -85,B 0,C 180,E1 3062.836,E2 3062.836} C_VEL
LIN {X 0,Y 148.632,Z 884.328,A -85,B 0,C 180,E1 3063.857,E2 3063.857} C_VEL
LIN {X 0,Y 139.491,Z 891.675,A -85,B 0,C 180,E1 3064.73,E2 3064.73} C_VEL
LIN {X 0,Y 133.974,Z 895.584,A -85,B 0,C 180,E1 3064.884,E2 3064.884} C_VEL
LIN {X 0,Y 126.341,Z 900.188,A -85,B 0,C 180,E1 3064.154,E2 3064.154} C_VEL
LIN {X 0,Y 119.208,Z 903.908,A -85,B 0,C 180,E1 3063.011,E2 3063.011} C_VEL
LIN {X 0,Y 103.528,Z 910.683,A -85,B 0,C 180,E1 3059.999,E2 3059.999} C_VEL
LIN {X 0,Y 88.187,Z 915.493,A -85,B 0,C 180,E1 3055.955,E2 3055.955} C_VEL
LIN {X 0,Y 73.053,Z 918.526,A -85,B 0,C 180,E1 3050.126,E2 3050.126} C_VEL
LIN {X 0,Y 58.212,Z 919.834,A -85,B 0,C 180,E1 3040.804,E2 3040.804} C_VEL
LIN {X 0,Y 46.41,Z 919.275,A -85,B 0,C 180,E1 3027.127,E2 3027.127} C_VEL
LIN {X 0,Y 38.235,Z 916.784,A -85,B 0,C 180,E1 3005.095,E2 3005.095} C_VEL
LIN {X 0,Y 37.005,Z 912.717,A -85,B 0,C 180,E1 2979.31,E2 2979.31} C_VEL
LIN {X 0,Y 42.055,Z 907.105,A -85,B 0,C 180,E1 2957.116,E2 2957.116} C_VEL
LIN {X 0,Y 51.555,Z 899.482,A -85,B 0,C 180,E1 2940.984,E2 2940.984} C_VEL
LIN {X 0,Y 62.211,Z 890.814,A -85,B 0,C 180,E1 2931.174,E2 2931.174} C_VEL
LIN {X 0,Y 73.132,Z 880.862,A -85,B 0,C 180,E1 2924.68,E2 2924.68} C_VEL
LIN {X 0,Y 84.628,Z 868.523,A -85,B 0,C 180,E1 2919.822,E2 2919.822} C_VEL
LIN {X 0,Y 95.101,Z 855.108,A -85,B 0,C 180,E1 2916.452,E2 2916.452} C_VEL
LIN {X 0,Y 103.89,Z 841.37,A -85,B 0,C 180,E1 2914.134,E2 2914.134} C_VEL
LIN {X 0,Y 111.827,Z 825.918,A -85,B 0,C 180,E1 2912.331,E2 2912.331} C_VEL
LIN {X 0,Y 118.368,Z 809.463,A -85,B 0,C 180,E1 2910.974,E2 2910.974} C_VEL
LIN {X 0,Y 123.18,Z 792.363,A -85,B 0,C 180,E1 2910.001,E2 2910.001} C_VEL
LIN {X 0,Y 126.345,Z 774.465,A -85,B 0,C 180,E1 2909.321,E2 2909.321} C_VEL
LIN {X 0,Y 134.218,Z 708.403,A -85,B 0,C 180,E1 2907.871,E2 2907.871} C_VEL
LIN {X 0,Y 133.28,Z 703.253,A -85,B 0,C 180,E1 2904.134,E2 2904.134} C_VEL
LIN {X 0,Y 132.665,Z 699.965,A -85,B 0,C 180,E1 2900.286,E2 2900.286} C_VEL
LIN {X 0,Y 132.448,Z 698.188,A -85,B 0,C 180,E1 2895.77,E2 2895.77} C_VEL
LIN {X 0,Y 132.828,Z 698.71,A -85,B 0,C 180,E1 2890.409,E2 2890.409} C_VEL
LIN {X 0,Y 133.484,Z 700.806,A -85,B 0,C 180,E1 2886.884,E2 2886.884} C_VEL
LIN {X 0,Y 134.447,Z 703.974,A -85,B 0,C 180,E1 2883.518,E2 2883.518} C_VEL
LIN {X 0,Y 135.462,Z 707.973,A -85,B 0,C 180,E1 2880.657,E2 2880.657} C_VEL
LIN {X 0,Y 125.908,Z 787.39,A -85,B 0,C 180,E1 2878.965,E2 2878.965} C_VEL
